// TwinCAT 3 PLC project PLC1
// ProgramVersion: 3.1.4023.0
// libraries:
//   CmpBitmapPool, * (System)
//   Tc2_MC2, * (Beckhoff Automation GmbH)
//   Tc2_Standard, * (Beckhoff Automation GmbH)
//   Tc2_System, * (Beckhoff Automation GmbH)
//   Tc2_Utilities, * (Beckhoff Automation GmbH)
//   Tc3_Module, * (Beckhoff Automation GmbH)
//   VisuDialogs, * (System)
//   VisuSymbols,3.5.10.0,System
// project tree:
//   DUTs/GVLs/ GVL.TcGVL, IOs.TcGVL
//   DUTs/ ST_CSV_Record.TcDUT
//   / GlobalTextList.TcGTLO, PlcTask.TcTTO, VISU_TASK.TcTTO
//   POUs/ Alarmes.TcPOU, InterfaceIOs.TcPOU, MAIN.TcPOU, CondicoesIniciais.TcPOU, IHM.TcPOU, Sinalizadores.TcPOU
//   POUs/Perifericos/ ReguaPotenciometrica.TcPOU, Robo.TcPOU, Inversores.TcPOU, Camera.TcPOU, MaquinaSolda.TcPOU, SafetyPLC.TcPOU, Servos.TcPOU, Valvulas.TcPOU
//   POUs/Receita/ Main_Receita.TcPOU, P_Read_Tabela.TcPOU, P_Write_Tabela.TcPOU
//   VISUs/ ImagePool.TcIPO (not stored), Lista_PontosSolda.TcVIS, Lista_PontosRoboCamera.TcVIS, Tela_Alarmes_2.TcVIS, Tela_Manual_2.TcVIS, Tela_Manual_3.TcVIS, Tela_Alarmes_1.TcVIS, Tela_Producao.TcVIS, Tela_Manual_1.TcVIS, Tela_Receita.TcVIS, Tela_Manutencao.TcVIS, VisualizationManager.TcVMO (not stored)

CONFIGURATION PLC1
    RESOURCE PLC ON TwinCAT3
        TASK PlcTask(INTERVAL := T#10ms, PRIORITY := 10);
        TASK VISU_TASK(INTERVAL := T#200000us, PRIORITY := 30);
        PROGRAM MAIN WITH PlcTask : MAIN;
        PROGRAM VisuElems_Visu_Prg WITH VISU_TASK : VisuElems.Visu_Prg;
    END_RESOURCE
END_CONFIGURATION

// ---- DUTs/ST_CSV_Record.TcDUT
TYPE ST_CSV_Record :
STRUCT
	sName 	: T_MaxString 	:= '';
	nNumber	: UDINT 		:= 0;
	fPos		: LREAL 		:= 0.0;
	bOP		: BOOL 		:= FALSE;
	sDesc		: STRING(40)	:= '';
	data		: ARRAY[0..7] OF BYTE;
END_STRUCT
END_TYPE

// ---- DUTs/GVLs/GVL.TcGVL
VAR_GLOBAL
(*========================================================================*)	

	FB_HoraAtual	: NT_GetTime;
	TempoAtual		: DT;
	Tempo_Atual_UTC	: DT;
	tempo			: TIMESTRUCT;
	
	MaquinaAlarme			: BOOL;
	MaquinaLigada			: BOOL;
	MaquinaModoManual		: BOOL;
	MaquinaModoAuto			: BOOL;
	Flag_CondicoesIniciais	: BOOL;
	Reset					: BOOL;

(*========================================================================*)

(*===================		ENTRADAS DIGITAIS		======================*)
	
	InMaquinaSolda_FK		: BOOL;
	InPinoCalha				: BOOL;
	InReset					: BOOL;
	InVermelho				: BOOL;
	InAmarelo				: BOOL;
	InVerde					: BOOL;
	InPecaOK				: BOOL;
	InSolda					: BOOL;
	
	//Sensores Fins de Curso
	InFimCurso1				: BOOL;
	InFimCurso2				: BOOL;
	InFimCurso3				: BOOL;
	InFimCurso4				: BOOL;

	//Sensores Painel Pneumático
	InPressostatoGeral		: BOOL;
	InSensorSegValvY7 		: BOOL;
	InSensorSegValvY8		: BOOL;
	
	//Sensores Indutivos
	InSensorIndutivo01		: BOOL;
	InSensorIndutivo02		: BOOL;
	InSensorIndutivo03		: BOOL;
	InSensorIndutivo04		: BOOL;
	InSensorIndutivo05		: BOOL;
	InSensorIndutivo06		: BOOL;
	InSensorIndutivo07		: BOOL;
	InSensorIndutivo08		: BOOL;
	InSensorIndutivo09		: BOOL;
	InSensorIndutivo10		: BOOL;
	InSensorIndutivo11		: BOOL;
	InSensorIndutivo12		: BOOL;
	
	//Comandos
	InComandoX				: BOOL;
	InComandoY				: BOOL;
	InComandoZ				: BOOL;
	InComando4				: BOOL;
	InComando5				: BOOL;
	InComando6				: BOOL;
	InComandoX1				: BOOL;
	InComandoX10			: BOOL;
	InComandoX100			: BOOL;
	InComandoStopC			: BOOL;
	InComandoStopCN			: BOOL;
	
	InSinalFaltaFase		: BOOL;
	InComandoPedal			: BOOL;
	InSolicitaEntrada		: BOOL;
	InSolicitaReset			: BOOL;
	
(*========================================================================*)

(*=====================		SAÍDAS DIGITAIS		==========================*)

	//Inversor 1 - Mesa Index
	OutLigarMesaIndex 			: BOOL;
	OutSentidoGiroMesaIndex 	: BOOL;
	
	//Inversor 2 - Esteira de Saída
	OutLigarEsteiraSaida		: BOOL;
	OutSentidoGiroEsteiraSaida	: BOOL;
	
	//Máquina de Solda
	OutMaquinaSolda_BtReset		: BOOL;
	OutMaquinaSolda_BtStart		: BOOL;
	
	OutMaquinaSolda_Receita_Bit1 : BOOL;
	OutMaquinaSolda_Receita_Bit2 : BOOL;
	OutMaquinaSolda_Receita_Bit3 : BOOL;
	OutMaquinaSolda_Receita_Bit4 : BOOL;
	OutMaquinaSolda_Receita_Bit5 : BOOL;
	
	//Válvulas
	OutValvulaY1A				: BOOL;
	OutValvulaY1R				: BOOL;
	OutValvulaY2A				: BOOL;
	OutValvulaY2R				: BOOL;
	OutValvulaY3A				: BOOL;
	OutValvulaY3R				: BOOL;
	OutValvulaY4A				: BOOL;
	OutValvulaY4R				: BOOL;
	OutValvulaY5A				: BOOL;
	OutValvulaY5R				: BOOL;
	OutValvulaY6				: BOOL;
	OutValvulaY7				: BOOL;
	OutValvulaY8				: BOOL;
	OutValvulaY9				: BOOL;
	
	//Sinalizadores Luminosos
	OutSinalizadorComandoLigado	: BOOL;
	OutSinalizadorBotoeiraHS1	: BOOL;
	OutSinalizadorBotoeiraHS2	: BOOL;
	
	//Sinalizador Luminoso - Manivela Eletrônica
	OutSinalizadorManivelaEletronica :BOOL;
	
(*========================================================================*)

(*=========================		SAFETY PLC		==========================*)	

	InSafety_CortinaLuz					: BOOL;
	InSafety_BtEmergenciaMaquinaSolda	: BOOL;
	InSafety_BtEmergenciaChiller		: BOOL;
	InSafety_BtEmergenciaRobo			: BOOL;
	InSafety_BtEmergenciaFrontal		: BOOL;
	InSafety_ChPortaMaquinaSolda		: BOOL;
	InSafety_ChPortaPainelPrincipal		: BOOL;
	InSafety_ChPortaEsteira				: BOOL;
	InSafety_ChPortaCamera				: BOOL;
	InSafety_ChPortaFrontalInferior		: BOOL;
	InSafety_ChPortaLateralEsquerdaFD	: BOOL;
	InSafety_ChPortaLateralEsquerdaFE	: BOOL;
	
	OutSafety_LiberacaoSDV1				: BOOL;
	OutSafety_ComandoSDV1				: BOOL;
	OutSafety_LiberacaoSDV2				: BOOL;
	OutSafety_ComandoSDV2				: BOOL;
	OutSafety_ComandoINVMesaIndex		: BOOL;
	OutSafety_ComandoINVEsteiraSaida	: BOOL;
	OutSafety_Comando1Robo				: BOOL;
	OutSafety_Comando2Robo				: BOOL;
	OutSafety_ParadaMaquinaSolda		: BOOL;
	OutSafety_SinalizacaoEmergencia		: BOOL;
	OutSafety_Reserva1					: BOOL;
	OutSafety_Reserva2					: BOOL;
	
	OutSafety_BtReset					: BOOL;
	
(*========================================================================*)

(*==========================		FLAG's		==========================*)	

	Flag_Maquina_MesaIndex			: BOOL;
	Flag_MesaIndex_Maquina			: BOOL;
	
	Flag_Maquina_EsteiraSaida		: BOOL;
	Flag_EsteiraSaida_Maquina		: BOOL;
	
	//Flag_Maquina_MaquinaSolda		: BOOL;
	//Flag_MaquinaSolda_Maquina		: BOOL;
	Flag_ServosXY_MaquinaSolda		: BOOL;
	Flag_MaquinaSolda_ServosXY		: BOOL;
	
	Flag_Maquina_Robo				: BOOL;
	Flag_Robo_Maquina				: BOOL;
	
	Flag_Robo_Camera				: BOOL;
	Flag_Camera_Robo				: BOOL;
	
	Flag_Maquina_ServosXY			: BOOL;
	Flag_ServosXY_Maquina			: BOOL;

(*========================================================================*)

(*=====================		MÁQUINA DE SOLDA		======================*)	

	LigarMaquinaSoldaManual			: BOOL;
	LigarMaquinaSoldaAuto			: BOOL;

(*========================================================================*)

(*=========================		CÂMERA SICK		==========================*)	

 Camera_Trigger					: BOOL;
 Camera_ChangeJob				: BOOL;
 Camera_SetJob					: BYTE;
 
 Camera_JobResult				: BOOL;
 Camera_JobCompleted			: BOOL;
 Camera_JobID					: BYTE;
 
 PecaAprovada					: BOOL;
 
 Camera_TargetJob				: ARRAY[0..5] OF INT;
 Camera_indexJob				: INT;
 
(*========================================================================*)

(*=========================		ROBÔ YASKAWA	==========================*)	

	Robot_CallMasterJob			: BOOL;
	Robot_ServoOn				: BOOL;
	Robot_ServoOff				: BOOL;
	Robot_ExtStart				: BOOL;
	Robot_ResetAlarm			: BOOL;
	
	Robot_HomePosition			: BOOL;
	Robot_TopMasterJob			: BOOL;
	Robot_AlarmStatus			: BOOL;
	
	
	Robot_IniciarCiclo			: BOOL;
	Robot_JobCompleted			: BOOL;
	Robot_JobCamera				: BOOL;
	
	Robot_NotSafetyPosition		: BOOL;
	
	Robot_Peca					: BOOL;
	Robot_Foto1					: BOOL;
	Robot_Foto2					: BOOL;

(*========================================================================*)

(*======================		SERVO MOTORES		======================*)	

	EixoX 							: AXIS_REF;
	EixoX_Energizado				: BOOL;
	
	EixoY 							: AXIS_REF;
	EixoY_Energizado				: BOOL;

(*========================================================================*)

(*=========================		INVERSORES		==========================*)	

	LigarMesaIndexAutomatico	: BOOL;
	LigarMesaIndexCiclo			: BOOL;
	LigarMesaIndexFwd			: BOOL;
	LigarMesaIndexBwd	 		: BOOL;
	LigarEsteiraSaidaFwd		: BOOL;
	LigarEsteiraSaidaBwd		: BOOL;
	
	FrequenciaMesaIndex			: REAL;
	FrequenciaEsteiraSaida		: REAL;
	
(*========================================================================*)
	
(*=========================		VÁLVULAS		==========================*)	

	AvancarValvulaY1			: BOOL;
	AvancarValvulaY2			: BOOL;
	AvancarValvulaY3			: BOOL;
	AvancarValvulaY4			: BOOL;
	AvancarValvulaY5			: BOOL;
	
	LigarValvulaY6				: BOOL;
	LigarValvulaY7				: BOOL;
	LigarValvulaY8				: BOOL;
	LigarValvulaY9				: BOOL;
	
	ValvulaProporcional			: REAL;
	
(*========================================================================*)

(*======================		ENTRADAS IHM		======================*)

	database_read					: ARRAY[0..MAX_CSV_ROWS, 0..MAX_CSV_COLUMNS ] OF STRING(MAX_CSV_FIELD_LENGTH);(* Target PLC database *)
	Simbolo_Atualizacao				: BOOL;

	b_selecionar_receita			: BOOL;
	b_deletar_receita				: BOOL;
	b_editar_receita				: BOOL;
	b_executar_receita				: BOOL;
	b_salvar_receita				: BOOL;
	b_cancelar_receita				: BOOL;
	b_criar_receita					: BOOL;
	bRead							: BOOL;
	bWrite							: BOOL;
	
(*======================		TELA RECEITA		======================*)

	//IhmEscr_Receita_MaquinaSolda		: INT;

(*======================		TELA MANUAL 1		======================*)
	//Controle da Máquina
	IhmBt_ManualAuto					: BOOL;
	IhmBt_ManualAuto_Text				: STRING;
	IhmBt_ManualAuto_Color				: BOOL;
		
	//ELEMENTOS PNEUMÁTICOS
	IhmBt_Y1_Ligar						: BOOL;
	IhmBt_Y2_Ligar						: BOOL;
	IhmBt_Y3_Ligar						: BOOL;
	IhmBt_Y4_Ligar						: BOOL;
	IhmBt_Y5_Ligar						: BOOL;
	
	IhmBt_Y6_Ligar						: BOOL;
	IhmBt_Y7_Ligar						: BOOL;
	IhmBt_Y8_Ligar						: BOOL;
	IhmBt_Y9_Ligar						: BOOL;	
	
	IhmBt_VP_Teste						: BOOL;
	
	//MOTORES
	//SERVO EIXO X E Y
	IhmBt_ServoXY_X1					: BOOL;
	IhmBt_ServoXY_X10					: BOOL;
	IhmBt_ServoXY_X100					: BOOL;
	
	//SERVO EIXO X
	IhmBt_ServoX_Reset					: BOOL;
	IhmBt_ServoX_Home					: BOOL;
	IhmBt_ServoX_JogBwd					: BOOL;
	IhmBt_ServoX_JogFwd					: BOOL;
	IhmBt_ServoX_PowerOn				: BOOL;
	IhmBt_ServoX_Referenciar			: BOOL;
	
	IhmLeit_ServoX_Posicao				: LREAL;
	IhmLeit_ServoX_Velocidade			: LREAL;
	IhmLeit_ServoX_Torque				: LREAL;
	
	//SERVO EIXO Y
	IhmBt_ServoY_Reset					: BOOL;
	IhmBt_ServoY_Home					: BOOL;
	IhmBt_ServoY_JogBwd					: BOOL;
	IhmBt_ServoY_JogFwd					: BOOL;
	IhmBt_ServoY_PowerOn				: BOOL;
	IhmBt_ServoY_Referenciar			: BOOL;
		
	IhmLeit_ServoY_Posicao				: LREAL;
	IhmLeit_ServoY_Velocidade			: LREAL;
	IhmLeit_ServoY_Torque				: LREAL;
	
	//INV. MESA INDEX
	IhmBt_MesaIndex_Sentido				: BOOL;
	IhmBt_MesaIndex_LigarDesligar		: BOOL;
	IhmBt_MesaIndex_Ciclo				: BOOL;
	
	//INV. ESTEIRA DE SAÍDA
	IhmBt_EsteiraSaida_Sentido			: BOOL;
	IhmBt_EsteiraSaida_LigarDesligar	: BOOL;
	
	IhmBt_MaquinaSolda_Reset			: BOOL;
	IhmBt_MaquinaSolda_Start			: BOOL;

(*======================		TELA MANUAL 2		======================*)
	
	IhmBt_ServoX_ReferenciarAutoINICIO				: BOOL;
	IhmBt_ServoX_ReferenciarAutoFIM					: BOOL;
	IhmBt_ServoY_ReferenciarAutoINICIO				: BOOL;
	IhmBt_ServoY_ReferenciarAutoFIM					: BOOL;
	
	IhmVs_PressaoPainelPneumatico_Text				: WSTRING;
	
	IhmBt_ReguaPotenciometrica_CalibrarRecuo		: BOOL;
	IhmBt_ReguaPotenciometrica_CalibrarPorca		: BOOL;
	IhmBt_ReguaPotenciometrica_CalibrarAvanco		: BOOL;
		
(*======================		TELA MANUAL 3		======================*)
	
	IhmBt_Camera_ChangeJob					: BOOL;
	IhmBt_Camera_Trigger					: BOOL;
	IhmLed_Camera_JobCompleted				: BOOL;
	IhmLed_Camera_JobResult					: BOOL;
	
	IhmLeit_Camera_JobID					: INT;
	
	IhmVs_Camera_JobResult_Text				: STRING;
		
(*========================================================================*)
	
	UserName		: STRING;
	UserGroupName	: STRING;
	UserGroupId		: DWORD;
	
	Blink_1hz		: BOOL;
	Blick_05hz		: BOOL;
	
	IhmBt_Ligar			: BOOL;
	IhmBt_Desligar		: BOOL;
	IhmBt_Reset			: BOOL;
	IhmBt_Pausar		: BOOL;
	IhmBt_CondIniciais	: BOOL;
	
	BT_ihm_zerar_contador	: BOOL;
	Contador_Total			: UDINT;
	Contador_PecasAprovadas	: UDINT;
	Contador_PecasReprovadas: UDINT;
	
	I1		: BOOL;
	I2		: BOOL;
	
	Recipe_Select_Int				: UDINT;
	Recipe_Names_Saved				: ARRAY [0..301] OF STRING;
	
	Recipe_Name_Select				: STRING;
	
	Recipe_No_Select				: INT;
	Recipe_ID_Select				: INT;
	
//	Recipe_Pos_HomeX_Select			: LREAL;
//	Recipe_Pos_HomeY_Select			: LREAL;
	
	Recipe_Pontos_Solda_Select		: INT;
	
	Recipe_P_X01_Solda_Select		: LREAL;
	Recipe_P_Y01_Solda_Select		: LREAL;
	Recipe_P01_Solda_Select			: BOOL;
	
	Recipe_P_X02_Solda_Select		: LREAL;
	Recipe_P_Y02_Solda_Select		: LREAL;
	Recipe_P02_Solda_Select			: BOOL;
	
	Recipe_P_X03_Solda_Select		: LREAL;
	Recipe_P_Y03_Solda_Select		: LREAL;
	Recipe_P03_Solda_Select			: BOOL;
	
	Recipe_P_X04_Solda_Select		: LREAL;
	Recipe_P_Y04_Solda_Select		: LREAL;
	Recipe_P04_Solda_Select			: BOOL;
	
	Recipe_P_X05_Solda_Select		: LREAL;
	Recipe_P_Y05_Solda_Select		: LREAL;
	Recipe_P05_Solda_Select			: BOOL;
	
	Recipe_P_X06_Solda_Select		: LREAL;
	Recipe_P_Y06_Solda_Select		: LREAL;
	Recipe_P06_Solda_Select			: BOOL;
	
	Recipe_P_X07_Solda_Select		: LREAL;
	Recipe_P_Y07_Solda_Select		: LREAL;
	Recipe_P07_Solda_Select			: BOOL;
	
	Recipe_P_X08_Solda_Select		: LREAL;
	Recipe_P_Y08_Solda_Select		: LREAL;
	Recipe_P08_Solda_Select			: BOOL;
	
	Recipe_P_X09_Solda_Select		: LREAL;
	Recipe_P_Y09_Solda_Select		: LREAL;
	Recipe_P09_Solda_Select			: BOOL;
	
	Recipe_P_X10_Solda_Select		: LREAL;
	Recipe_P_Y10_Solda_Select		: LREAL;
	Recipe_P10_Solda_Select			: BOOL;
	
	Recipe_P_X11_Solda_Select		: LREAL;
	Recipe_P_Y11_Solda_Select		: LREAL;
	Recipe_P11_Solda_Select			: BOOL;
	
	Recipe_P_X12_Solda_Select		: LREAL;
	Recipe_P_Y12_Solda_Select		: LREAL;
	Recipe_P12_Solda_Select			: BOOL;
	
	Recipe_P_X13_Solda_Select		: LREAL;
	Recipe_P_Y13_Solda_Select		: LREAL;
	Recipe_P13_Solda_Select			: BOOL;
	
	Recipe_P_X14_Solda_Select		: LREAL;
	Recipe_P_Y14_Solda_Select		: LREAL;
	Recipe_P14_Solda_Select			: BOOL;
	
	Recipe_P_X15_Solda_Select		: LREAL;
	Recipe_P_Y15_Solda_Select		: LREAL;
	Recipe_P15_Solda_Select			: BOOL;

	Recipe_Pontos_Camera_Select		: INT;
	Recipe_JobID_F01_Camera_Select	: INT;
	Recipe_JobID_F02_Camera_Select	: INT;
	Recipe_JobID_F03_Camera_Select	: INT;
	Recipe_JobID_F04_Camera_Select	: INT;
	Recipe_JobID_F05_Camera_Select	: INT;
	
//	Recipe_F01_Camera_Select		: BOOL;
//	Recipe_F02_Camera_Select		: BOOL;
//	Recipe_F03_Camera_Select		: BOOL;
//	Recipe_F04_Camera_Select		: BOOL;
//	Recipe_F05_Camera_Select		: BOOL;


	Recipe_Valvula_Proporcional_Select	: LREAL;
	
	Recipe_Pecas_Caixa_Select		: INT;
		
	NumPontosSolda					: INT;
	NumPontosCamera					: INT;
	
	TargetX							: ARRAY[0..14] OF LREAL;
	TargetY							: ARRAY[0..14] OF LREAL;
	SoldaXY							: ARRAY[0..14] OF BOOL;
	
	CameraJobID						: ARRAY[0..4] OF INT;
	
	PosicaoOrigemX					: LREAL;
	PosicaoOrigemY					: LREAL;
	
(*========================================================================*)
	
END_VAR

VAR_GLOBAL RETAIN

(*======================		TELA RECEITA		======================*)

	IhmEscr_Receita_MaquinaSolda		: INT;

(*======================		TELA MANUAL 1		======================*)

	//ELEMENTOS PNEUMÁTICOS
	IhmEscr_ValvulaProporcional			: INT;

	//SERVO EIXO X E Y
	IhmEscr_ServoXY_TorqueMax			: INT;
	IhmEscr_ServoXY_TempoTorqueMax		: INT;
	IhmEscr_ServoXY_VelocidadeAuto		: INT;
	IhmEscr_ServoXY_VelocidadeManual	: INT;
	
	//INV. MESA INDEX
	IhmEscr_MesaIndex_Frequencia		: INT;
	IhmEscr_MesaIndex_DelayParada		: REAL;
	
	//INV. ESTEIRA DE SAÍDA
	IhmEscr_EsteiraSaida_Frequencia		: INT;

(*======================		TELA MANUAL 2		======================*)
	
	IhmEscr_ReguaPotenciometrica_ToleranciaRecuo	: REAL;
	IhmEscr_ReguaPotenciometrica_ToleranciaPorca	: REAL;
	IhmEscr_ReguaPotenciometrica_ToleranciaAvanco	: REAL;	
		
(*======================		TELA MANUAL 3		======================*)
	
	IhmEscr_Camera_SetJob					: INT;
	
	IhmEscr_Camera_DelayError				: TIME;
	
(*==================		RÉGUA POTENCIOMÉTRICA		==================*)	

	ReguaPotenciometricaPosicao			: REAL;
	ReguaPotenciometricaSinal			: INT;
	
	ReguaPotenciometrica_Recuada		: REAL;
	ReguaPotenciometrica_Recuada_LI		: REAL;
	ReguaPotenciometrica_Recuada_LS		: REAL;

	ReguaPotenciometrica_Porca			: REAL;
	ReguaPotenciometrica_Porca_LI		: REAL;
	ReguaPotenciometrica_Porca_LS		: REAL;

	ReguaPotenciometrica_Avancada		: REAL;
	ReguaPotenciometrica_Avancada_LI	: REAL;
	ReguaPotenciometrica_Avancada_LS	: REAL;
	
(*========================================================================*)

END_VAR

VAR_GLOBAL CONSTANT

	MAX_CSV_ROWS 			: UDINT := 30;
	MAX_CSV_COLUMNS 		: UDINT := 60;
	MAX_CSV_FIELD_LENGTH	: UDINT := 100;

END_VAR

// ---- DUTs/GVLs/IOs.TcGVL
VAR_GLOBAL

(*======================		ENTRADAS DIGITAIS		======================*)

	//Cartão de Entradas 0:= EntradaI0_0
	EntradaI0_0		AT %I*	: BOOL;
	EntradaI0_1		AT %I*	: BOOL;
	EntradaI0_2		AT %I*	: BOOL;
	EntradaI0_3		AT %I*	: BOOL;
	EntradaI0_4		AT %I*	: BOOL;
	EntradaI0_5		AT %I*	: BOOL;
	EntradaI0_6		AT %I*	: BOOL;
	EntradaI0_7		AT %I*	: BOOL;
	EntradaI1_0		AT %I*	: BOOL;
	EntradaI1_1		AT %I*	: BOOL;
	EntradaI1_2		AT %I*	: BOOL;
	EntradaI1_3		AT %I*	: BOOL;
	EntradaI1_4		AT %I*	: BOOL;
	EntradaI1_5		AT %I*	: BOOL;
	EntradaI1_6		AT %I*	: BOOL;
	EntradaI1_7		AT %I*	: BOOL;
	
	//Cartão de Entradas 1
	EntradaI2_0		AT %I*	: BOOL;
	EntradaI2_1		AT %I*	: BOOL;
	EntradaI2_2		AT %I*	: BOOL;
	EntradaI2_3		AT %I*	: BOOL;
	EntradaI2_4		AT %I*	: BOOL;
	EntradaI2_5		AT %I*	: BOOL;
	EntradaI2_6		AT %I*	: BOOL;
	EntradaI2_7		AT %I*	: BOOL;
	EntradaI3_0		AT %I*	: BOOL;
	EntradaI3_1		AT %I*	: BOOL;
	EntradaI3_2		AT %I*	: BOOL;
	EntradaI3_3		AT %I*	: BOOL;
	EntradaI3_4		AT %I*	: BOOL;
	EntradaI3_5		AT %I*	: BOOL;
	EntradaI3_6		AT %I*	: BOOL;
	EntradaI3_7		AT %I*	: BOOL;
	
	//Cartão de Entradas 2
	EntradaI4_0		AT %I*	: BOOL;
	EntradaI4_1		AT %I*	: BOOL;
	EntradaI4_2		AT %I*	: BOOL;
	EntradaI4_3		AT %I*	: BOOL;
	EntradaI4_4		AT %I*	: BOOL;
	EntradaI4_5		AT %I*	: BOOL;
	EntradaI4_6		AT %I*	: BOOL;
	EntradaI4_7		AT %I*	: BOOL;
	EntradaI5_0		AT %I*	: BOOL;
	EntradaI5_1		AT %I*	: BOOL;
	EntradaI5_2		AT %I*	: BOOL;
	EntradaI5_3		AT %I*	: BOOL;
	EntradaI5_4		AT %I*	: BOOL;
	EntradaI5_5		AT %I*	: BOOL;
	EntradaI5_6		AT %I*	: BOOL;
	EntradaI5_7		AT %I*	: BOOL;
	
	//Cartão de Entradas 3
	EntradaI6_0		AT %I*	: BOOL;
	EntradaI6_1		AT %I*	: BOOL;
	EntradaI6_2		AT %I*	: BOOL;
	EntradaI6_3		AT %I*	: BOOL;
	EntradaI6_4		AT %I*	: BOOL;
	EntradaI6_5		AT %I*	: BOOL;
	EntradaI6_6		AT %I*	: BOOL;
	EntradaI6_7		AT %I*	: BOOL;
	EntradaI7_0		AT %I*	: BOOL;
	EntradaI7_1		AT %I*	: BOOL;
	EntradaI7_2		AT %I*	: BOOL;
	EntradaI7_3		AT %I*	: BOOL;
	EntradaI7_4		AT %I*	: BOOL;
	EntradaI7_5		AT %I*	: BOOL;
	EntradaI7_6		AT %I*	: BOOL;
	EntradaI7_7		AT %I*	: BOOL;
	
(*============================================================================*)
(*=========================		SAÍDAS DIGITAIS		==========================*)
	//Outputs
	
	//Cartão de Saídas 0
	SaidaQ0_0		AT %Q*	: BOOL;
	SaidaQ0_1		AT %Q*	: BOOL;
	SaidaQ0_2		AT %Q*	: BOOL;
	SaidaQ0_3		AT %Q*	: BOOL;
	SaidaQ0_4		AT %Q*	: BOOL;
	SaidaQ0_5		AT %Q*	: BOOL;
	SaidaQ0_6		AT %Q*	: BOOL;
	SaidaQ0_7		AT %Q*	: BOOL;
	SaidaQ1_0		AT %Q*	: BOOL;
	SaidaQ1_1		AT %Q*	: BOOL;
	SaidaQ1_2		AT %Q*	: BOOL;
	SaidaQ1_3		AT %Q*	: BOOL;
	SaidaQ1_4		AT %Q*	: BOOL;
	SaidaQ1_5		AT %Q*	: BOOL;
	SaidaQ1_6		AT %Q*	: BOOL;
	SaidaQ1_7		AT %Q*	: BOOL;
	
	//Cartão de Saídas 1
	SaidaQ2_0		AT %Q*	: BOOL;
	SaidaQ2_1		AT %Q*	: BOOL;
	SaidaQ2_2		AT %Q*	: BOOL;
	SaidaQ2_3		AT %Q*	: BOOL;
	SaidaQ2_4		AT %Q*	: BOOL;
	SaidaQ2_5		AT %Q*	: BOOL;
	SaidaQ2_6		AT %Q*	: BOOL;
	SaidaQ2_7		AT %Q*	: BOOL;
	SaidaQ3_0		AT %Q*	: BOOL;
	SaidaQ3_1		AT %Q*	: BOOL;
	SaidaQ3_2		AT %Q*	: BOOL;
	SaidaQ3_3		AT %Q*	: BOOL;
	SaidaQ3_4		AT %Q*	: BOOL;
	SaidaQ3_5		AT %Q*	: BOOL;
	SaidaQ3_6		AT %Q*	: BOOL;
	SaidaQ3_7		AT %Q*	: BOOL;
	
	//Cartão de Saídas 2
	SaidaQ4_0		AT %Q*	: BOOL;
	SaidaQ4_1		AT %Q*	: BOOL;
	SaidaQ4_2		AT %Q*	: BOOL;
	SaidaQ4_3		AT %Q*	: BOOL;
	SaidaQ4_4		AT %Q*	: BOOL;
	SaidaQ4_5		AT %Q*	: BOOL;
	SaidaQ4_6		AT %Q*	: BOOL;
	SaidaQ4_7		AT %Q*	: BOOL;
	SaidaQ5_0		AT %Q*	: BOOL;
	SaidaQ5_1		AT %Q*	: BOOL;
	SaidaQ5_2		AT %Q*	: BOOL;
	SaidaQ5_3		AT %Q*	: BOOL;
	SaidaQ5_4		AT %Q*	: BOOL;
	SaidaQ5_5		AT %Q*	: BOOL;
	SaidaQ5_6		AT %Q*	: BOOL;
	SaidaQ5_7		AT %Q*	: BOOL;
	
	//Cartão de Saídas 3
	SaidaQ6_0		AT %Q*	: BOOL;
	SaidaQ6_1		AT %Q*	: BOOL;
	SaidaQ6_2		AT %Q*	: BOOL;
	SaidaQ6_3		AT %Q*	: BOOL;
	SaidaQ6_4		AT %Q*	: BOOL;
	SaidaQ6_5		AT %Q*	: BOOL;
	SaidaQ6_6		AT %Q*	: BOOL;
	SaidaQ6_7		AT %Q*	: BOOL;
	SaidaQ7_0		AT %Q*	: BOOL;
	SaidaQ7_1		AT %Q*	: BOOL;
	SaidaQ7_2		AT %Q*	: BOOL;
	SaidaQ7_3		AT %Q*	: BOOL;
	SaidaQ7_4		AT %Q*	: BOOL;
	SaidaQ7_5		AT %Q*	: BOOL;
	SaidaQ7_6		AT %Q*	: BOOL;
	SaidaQ7_7		AT %Q*	: BOOL;	

(*============================================================================*)
(*======================		ENTRADAS ANALÓGICAS		======================*)

	//Cartão de Entradas
	EntradaA0_0		AT %I*	: INT;
	EntradaA0_1		AT %I*	: INT;
	EntradaA0_2		AT %I*	: INT;
	EntradaA0_3		AT %I*	: INT;

(*============================================================================*)	
	
(*============================================================================*)
(*======================		SAÍDAS ANALÓGICAS		======================*)

	//Cartão de Saídas 0
	SaidaA0_0		AT %Q*	: INT;
	SaidaA0_1		AT %Q*	: INT;
	SaidaA0_2		AT %Q*	: INT;
	SaidaA0_3		AT %Q*	: INT;
		
(*============================================================================*)

(*======================		REDE ETHERNET/IP		======================*)

(*==========================		SAFETY PLC		==========================*)

	SafetyPLC_In_Byte0 		AT %I*:BYTE;
	SafetyPLC_In_Byte1 		AT %I*:BYTE;
	SafetyPLC_In_Byte2 		AT %I*:BYTE;
	SafetyPLC_In_Byte3 		AT %I*:BYTE;
	SafetyPLC_In_Byte4 		AT %I*:BYTE;
	SafetyPLC_In_Byte5 		AT %I*:BYTE;
	
	SafetyPLC_Out_Byte0 	AT %Q*:BYTE;

(*============================================================================*)

(*===================		CÂMERA SICK - INSPECTOR 63		==================*)

	CameraSickIn_0		AT %I*:BYTE;
	CameraSickIn_1		AT %I*:BYTE;
	CameraSickIn_2		AT %I*:BYTE;
	CameraSickIn_3		AT %I*:BYTE;
	CameraSickIn_4		AT %I*:BYTE;
	CameraSickIn_5		AT %I*:BYTE;
	CameraSickIn_6		AT %I*:BYTE;
	CameraSickIn_7		AT %I*:BYTE;
	CameraSickIn_8		AT %I*:BYTE;
	CameraSickIn_9		AT %I*:BYTE;

	CameraSickOut_0		AT %Q*:BYTE;
	CameraSickOut_1		AT %Q*:BYTE;
	CameraSickOut_2		AT %Q*:BYTE;
	CameraSickOut_3		AT %Q*:BYTE;
	CameraSickOut_4		AT %Q*:BYTE;
	CameraSickOut_5		AT %Q*:BYTE;
	CameraSickOut_6		AT %Q*:BYTE;
	CameraSickOut_7		AT %Q*:BYTE;
	CameraSickOut_8		AT %Q*:BYTE;
	CameraSickOut_9		AT %Q*:BYTE;

(*============================================================================*)

(*=====================		ROBÔ YASKAWA/MOTOMAN		======================*)
	
	Robot_PLC_0 		AT %I*:BYTE;
	Robot_PLC_1 		AT %I*:BYTE;
	Robot_PLC_2 		AT %I*:BYTE;
	Robot_PLC_3 		AT %I*:BYTE;
	Robot_PLC_4 		AT %I*:BYTE;
	Robot_PLC_5 		AT %I*:BYTE;
	Robot_PLC_6 		AT %I*:BYTE;
	Robot_PLC_7 		AT %I*:BYTE;
	Robot_PLC_8 		AT %I*:BYTE;
	Robot_PLC_9 		AT %I*:BYTE;
	Robot_PLC_10 		AT %I*:BYTE;
	Robot_PLC_11 		AT %I*:BYTE;
	Robot_PLC_12 		AT %I*:BYTE;
	Robot_PLC_13 		AT %I*:BYTE;
	Robot_PLC_14 		AT %I*:BYTE;
	Robot_PLC_15 		AT %I*:BYTE;
	Robot_PLC_16 		AT %I*:BYTE;
	Robot_PLC_17 		AT %I*:BYTE;
	Robot_PLC_18 		AT %I*:BYTE;
	Robot_PLC_19 		AT %I*:BYTE;
	
	PLC_Robot_0			AT %Q*:BYTE;
	PLC_Robot_1			AT %Q*:BYTE;
	PLC_Robot_2			AT %Q*:BYTE;
	PLC_Robot_3			AT %Q*:BYTE;
	PLC_Robot_4			AT %Q*:BYTE;
	PLC_Robot_5			AT %Q*:BYTE;
	PLC_Robot_6			AT %Q*:BYTE;
	PLC_Robot_7			AT %Q*:BYTE;
	PLC_Robot_8			AT %Q*:BYTE;
	PLC_Robot_9			AT %Q*:BYTE;
	PLC_Robot_10		AT %Q*:BYTE;
	PLC_Robot_11		AT %Q*:BYTE;
	PLC_Robot_12		AT %Q*:BYTE;
	PLC_Robot_13		AT %Q*:BYTE;
	PLC_Robot_14		AT %Q*:BYTE;
	PLC_Robot_15		AT %Q*:BYTE;

(*============================================================================*)
	
END_VAR

// ---- POUs/MAIN.TcPOU
PROGRAM MAIN
VAR
		
	SafetyPLCIn 	AT %I*:BYTE;
	SafetyPLCOut 	AT %Q*:BYTE;
	
	sUrlAddressCamera : STRING;

	writeData:FB_WritePersistentData;
	t1:TON;
	bSavePersistent: BOOL;
	
	timer_login	: TON;
	
	Timer_Blink_1hz_1	: TON;
	Timer_Blink_1hz_2	: TON;
	
	b_contador		: BOOL;
	int_contador_10		: INT;
	
	
	PassoBtLigarDesligar	: INT;
	PassoBtReset			: INT;
	PassoMaquina			: INT;
	
END_VAR

(*=====================		ROTINAS EXECUTADAS		======================*)

Main_Receita();
CondicoesIniciais();
Alarmes();
InterfaceIOs();
Inversores();
Valvulas();
ReguaPotenciometrica();
Servos();
Robo();
Camera();
MaquinaSolda();
IHM();
Sinalizadores();

(*=================		INTERFACE CÂMERA SICK		======================*)

sUrlAddressCamera := 'http://192.168.10.20/';

(*=====================		ROTINA PRINCIPAL		======================*)	

//Condição de Bloqueio da Máquina de Estados - Mesa Index FWD
IF (Alarmes.AlarmeGrave
	//OR Alarmes.AlarmeMedio
	//OR Alarmes.AlarmeLeve
	OR NOT MaquinaLigada
	OR NOT MaquinaModoAuto
	) THEN
	PassoMaquina := 1000;
	MaquinaLigada := FALSE;
	Flag_Maquina_MesaIndex := FALSE;
	Flag_Maquina_ServosXY := FALSE;	
	Flag_Maquina_Robo := FALSE;
	Flag_Maquina_EsteiraSaida := FALSE;
END_IF

CASE PassoMaquina OF

	//Passo 0 - Inicialização
	0: PassoMaquina := 10;
	
	//Passo 10 - Verificar condições iniciais
	10: PassoMaquina := 20;
	
	//Passo 20 - Comando para iniciar ciclo 
	20: //IF InComandoPedal THEN
			PassoMaquina := 30;
		//END_IF
	
	//Passo 30 - Dar Passo na Mesa Index
	30: Flag_Maquina_MesaIndex := TRUE;
		PassoMaquina := 40;
		
	//Passo 40 - Verificar Conclusão do Movimento da Mesa Index
	40: IF Flag_MesaIndex_Maquina THEN
			Flag_MesaIndex_Maquina := FALSE;
			PassoMaquina := 50;
		END_IF
		
	//Passo 50 - Liberar Servos XY
	50: Flag_Maquina_ServosXY := TRUE;
		PassoMaquina := 60;
		
	//Passo 60 - Liberar Ação do Robô
	60: Flag_Maquina_Robo := TRUE;
		PassoMaquina := 70;
		
	//Passo 70 - Verificar Conclusão da Rotina dos Servos e da Máquina de Solda
	70: IF Flag_ServosXY_Maquina THEN
			Flag_ServosXY_Maquina := FALSE;
			PassoMaquina := 80;
		END_IF
	
	//Passo 80 - Verificar Conclusão da Rotina Avaliação da Peça (Robô e Câmera)
	80: IF Flag_Robo_Maquina THEN
			Flag_Robo_Maquina := FALSE;
			PassoMaquina := 1000;
		END_IF
	
	//Passo 1000 - Finalização
	1000: PassoMaquina := 0;

END_CASE

(*========================================================================*)

END_PROGRAM

// ---- POUs/Receita/Main_Receita.TcPOU
PROGRAM Main_Receita
VAR
	(*	In USA/UK the CSV field separator is a comma.
	In Germany and some other European countries the CSV field separator is a semicolon. *)
	bChangeSeparatorToComma	: BOOL := FALSE;
	
	i : UDINT;
	
	PassoLimparMemoriasReceita 	: INT;
	
	timer_Leitura_Receitas_Salvas	: TON;
	Endereco_vazio		: INT;
	b_reorganizar		: INT;
	Item_deletado		: UDINT;
	Item_criar			: UDINT;
	Item_livre			: UDINT;
	Item_Atual			: UDINT;
	
	Row_copy			: ARRAY[0..MAX_CSV_COLUMNS] OF STRING(MAX_CSV_FIELD_LENGTH);(* Target PLC database *)
	
	LengthScrollBar_PontosSolda			: INT;
	ScrollBar_PontosSolda				: INT;
	ScrollScreen_PontosSolda			: INT;
	
	LengthScrollBar_PontosCamera		: INT;
	ScrollBar_PontosCamera				: INT;
	ScrollScreen_PontosCamera			: INT;
	
END_VAR

(*========================================================================*)
(*=============		BARRA DE ROLAGEM - TELA RECEITAS		==============*)

//Lista de Pontos de Solda
IF(Recipe_Pontos_Solda_Select <=2) THEN
	ScrollBar_PontosSolda := 0;
	LengthScrollBar_PontosSolda := 0;
ELSE
	LengthScrollBar_PontosSolda := (Recipe_Pontos_Solda_Select-2)*60;
END_IF

ScrollScreen_PontosSolda := (-1)*ScrollBar_PontosSolda;

//Lista de Pontos de Avaliação - Câmera
IF(Recipe_Pontos_Camera_Select <=2) THEN
	ScrollBar_PontosCamera := 0;
	LengthScrollBar_PontosCamera := 0;
ELSE
	LengthScrollBar_PontosCamera := (Recipe_Pontos_Camera_Select-2)*60;
END_IF

ScrollScreen_PontosCamera := (-1)*ScrollBar_PontosCamera;

(*========================================================================*)

IF bChangeSeparatorToComma THEN
	DEFAULT_CSV_FIELD_SEP := 16#2C;(* Comma ASCII code *)
ELSE
	DEFAULT_CSV_FIELD_SEP := 16#3B;(* Semicolon ASCII code *)
END_IF

P_Read_Tabela();
P_Write_Tabela();
//P_ArgToConvExample();(* This sample program shows the usage of the ARG_TO_CSVFIELD and CSVFILED_TO_ARG conversion functions *)
//P_StringToConvExample(); (* This sample program shows the usage of the STRING_TO_CSVFIELD and CSVFIELD_TO_STRING conversion functions *)

(*timer_Leitura_Receitas_Salvas (in := TRUE, pt := T#1M);
IF timer_Leitura_Receitas_Salvas.Q THEN
	timer_Leitura_Receitas_Salvas (in := FALSE);
	bRead := TRUE;
END_IF*)

IF NOT b_deletar_receita AND NOT b_editar_receita AND NOT b_criar_receita THEN
	
	Recipe_Name_Select					:= database_read[Recipe_select_int, 0];
	Recipe_No_Select					:= STRING_TO_INT	(database_read[Recipe_select_int, 1]);
	Recipe_ID_Select					:= STRING_TO_INT	(database_read[Recipe_select_int, 2]);
		
	Recipe_Pontos_Solda_Select			:= STRING_TO_INT	(database_read[Recipe_select_int, 3]);
		
	Recipe_P_X01_Solda_Select			:= STRING_TO_LREAL 	(database_read[Recipe_select_int, 4]);
	Recipe_P_Y01_Solda_Select			:= STRING_TO_LREAL 	(database_read[Recipe_select_int, 5]);
	Recipe_P01_Solda_Select				:= STRING_TO_BOOL	(database_read[Recipe_select_int, 6]);
	Recipe_P_X02_Solda_Select			:= STRING_TO_LREAL 	(database_read[Recipe_select_int, 7]);
	Recipe_P_Y02_Solda_Select			:= STRING_TO_LREAL 	(database_read[Recipe_select_int, 8]);
	Recipe_P02_Solda_Select				:= STRING_TO_BOOL	(database_read[Recipe_select_int, 9]);	
	Recipe_P_X03_Solda_Select			:= STRING_TO_LREAL 	(database_read[Recipe_select_int, 10]);
	Recipe_P_Y03_Solda_Select			:= STRING_TO_LREAL 	(database_read[Recipe_select_int, 11]);
	Recipe_P03_Solda_Select				:= STRING_TO_BOOL	(database_read[Recipe_select_int, 12]);
	Recipe_P_X04_Solda_Select			:= STRING_TO_LREAL 	(database_read[Recipe_select_int, 13]);
	Recipe_P_Y04_Solda_Select			:= STRING_TO_LREAL 	(database_read[Recipe_select_int, 14]);
	Recipe_P04_Solda_Select				:= STRING_TO_BOOL	(database_read[Recipe_select_int, 15]);
	Recipe_P_X05_Solda_Select			:= STRING_TO_LREAL 	(database_read[Recipe_select_int, 16]);
	Recipe_P_Y05_Solda_Select			:= STRING_TO_LREAL 	(database_read[Recipe_select_int, 17]);
	Recipe_P05_Solda_Select				:= STRING_TO_BOOL	(database_read[Recipe_select_int, 18]);
	
	Recipe_P_X06_Solda_Select			:= STRING_TO_LREAL 	(database_read[Recipe_select_int, 19]);
	Recipe_P_Y06_Solda_Select			:= STRING_TO_LREAL 	(database_read[Recipe_select_int, 20]);
	Recipe_P06_Solda_Select				:= STRING_TO_BOOL	(database_read[Recipe_select_int, 21]);
	Recipe_P_X07_Solda_Select			:= STRING_TO_LREAL 	(database_read[Recipe_select_int, 22]);
	Recipe_P_Y07_Solda_Select			:= STRING_TO_LREAL 	(database_read[Recipe_select_int, 23]);
	Recipe_P07_Solda_Select				:= STRING_TO_BOOL	(database_read[Recipe_select_int, 24]);	
	Recipe_P_X08_Solda_Select			:= STRING_TO_LREAL 	(database_read[Recipe_select_int, 25]);
	Recipe_P_Y08_Solda_Select			:= STRING_TO_LREAL 	(database_read[Recipe_select_int, 26]);
	Recipe_P08_Solda_Select				:= STRING_TO_BOOL	(database_read[Recipe_select_int, 27]);
	Recipe_P_X09_Solda_Select			:= STRING_TO_LREAL 	(database_read[Recipe_select_int, 28]);
	Recipe_P_Y09_Solda_Select			:= STRING_TO_LREAL 	(database_read[Recipe_select_int, 29]);
	Recipe_P09_Solda_Select				:= STRING_TO_BOOL	(database_read[Recipe_select_int, 30]);
	Recipe_P_X10_Solda_Select			:= STRING_TO_LREAL 	(database_read[Recipe_select_int, 31]);
	Recipe_P_Y10_Solda_Select			:= STRING_TO_LREAL 	(database_read[Recipe_select_int, 32]);
	Recipe_P10_Solda_Select				:= STRING_TO_BOOL	(database_read[Recipe_select_int, 33]);
		
	Recipe_P_X11_Solda_Select			:= STRING_TO_LREAL 	(database_read[Recipe_select_int, 34]);
	Recipe_P_Y11_Solda_Select			:= STRING_TO_LREAL 	(database_read[Recipe_select_int, 35]);
	Recipe_P11_Solda_Select				:= STRING_TO_BOOL	(database_read[Recipe_select_int, 36]);
	Recipe_P_X12_Solda_Select			:= STRING_TO_LREAL 	(database_read[Recipe_select_int, 37]);
	Recipe_P_Y12_Solda_Select			:= STRING_TO_LREAL 	(database_read[Recipe_select_int, 38]);
	Recipe_P12_Solda_Select				:= STRING_TO_BOOL	(database_read[Recipe_select_int, 39]);	
	Recipe_P_X13_Solda_Select			:= STRING_TO_LREAL 	(database_read[Recipe_select_int, 40]);
	Recipe_P_Y13_Solda_Select			:= STRING_TO_LREAL 	(database_read[Recipe_select_int, 41]);
	Recipe_P13_Solda_Select				:= STRING_TO_BOOL	(database_read[Recipe_select_int, 42]);
	Recipe_P_X14_Solda_Select			:= STRING_TO_LREAL 	(database_read[Recipe_select_int, 43]);
	Recipe_P_Y14_Solda_Select			:= STRING_TO_LREAL 	(database_read[Recipe_select_int, 44]);
	Recipe_P14_Solda_Select				:= STRING_TO_BOOL	(database_read[Recipe_select_int, 45]);
	Recipe_P_X15_Solda_Select			:= STRING_TO_LREAL 	(database_read[Recipe_select_int, 46]);
	Recipe_P_Y15_Solda_Select			:= STRING_TO_LREAL 	(database_read[Recipe_select_int, 47]);
	Recipe_P15_Solda_Select				:= STRING_TO_BOOL	(database_read[Recipe_select_int, 48]);
		
	Recipe_Valvula_Proporcional_Select	:= STRING_TO_LREAL 	(database_read[Recipe_select_int, 49]);
	
	Recipe_Pontos_Camera_Select			:= STRING_TO_INT	(database_read[Recipe_select_int, 50]);
	Recipe_JobID_F01_Camera_Select		:= STRING_TO_INT 	(database_read[Recipe_select_int, 51]);
	Recipe_JobID_F02_Camera_Select		:= STRING_TO_INT 	(database_read[Recipe_select_int, 52]);
	Recipe_JobID_F03_Camera_Select		:= STRING_TO_INT 	(database_read[Recipe_select_int, 53]);
	Recipe_JobID_F04_Camera_Select		:= STRING_TO_INT 	(database_read[Recipe_select_int, 54]);
	Recipe_JobID_F05_Camera_Select		:= STRING_TO_INT 	(database_read[Recipe_select_int, 55]);

	Recipe_Pecas_Caixa_Select			:= STRING_TO_INT 	(database_read[Recipe_select_int, 56]);
	
	Recipe_names_saved [i] := database_read [i,0];

	IF Recipe_names_saved[i] <> '' THEN
		Item_Atual := 1;	
	END_IF
	
	IF Item_Atual = 1 AND Recipe_names_saved[i] = '' THEN
		Item_Atual := 0;
		Item_livre := i;
		i:=0; 
	END_IF
	
	i := i +1;
	IF (i >= MAX_CSV_ROWS)  THEN 
		i:=0; 
	END_IF
END_IF
	
// Verificações
//	Ao Deletar e salvar uma receita - O sistema deve verificar qual endereço ficou em vazio, e fazer uma rotina de reorganiza-lo e depois escrever na tabela de receitas
// Criar Receitar - verificar qual o ultima endereço da tabela vazia. Escrever ali o valores e ao apertar salvar escrever na tabela de receitas
//Editar e Cancelar - Não escreve na tabela

IF b_deletar_receita AND b_reorganizar = 0 THEN
	
	Recipe_Name_Select					:= '';
	Recipe_No_Select					:= 0;
	Recipe_ID_Select					:= 0;
		
	Recipe_Pontos_Solda_Select			:= 0;
		
	Recipe_P_X01_Solda_Select			:= 0.0;
	Recipe_P_Y01_Solda_Select			:= 0.0;
	Recipe_P01_Solda_Select				:= FALSE;
	Recipe_P_X02_Solda_Select			:= 0.0;
	Recipe_P_Y02_Solda_Select			:= 0.0;
	Recipe_P02_Solda_Select				:= FALSE;	
	Recipe_P_X03_Solda_Select			:= 0.0;
	Recipe_P_Y03_Solda_Select			:= 0.0;
	Recipe_P03_Solda_Select				:= FALSE;
	Recipe_P_X04_Solda_Select			:= 0.0;
	Recipe_P_Y04_Solda_Select			:= 0.0;
	Recipe_P04_Solda_Select				:= FALSE;
	Recipe_P_X05_Solda_Select			:= 0.0;
	Recipe_P_Y05_Solda_Select			:= 0.0;
	Recipe_P05_Solda_Select				:= FALSE;
	
	Recipe_P_X06_Solda_Select			:= 0.0;
	Recipe_P_Y06_Solda_Select			:= 0.0;
	Recipe_P06_Solda_Select				:= FALSE;
	Recipe_P_X07_Solda_Select			:= 0.0;
	Recipe_P_Y07_Solda_Select			:= 0.0;
	Recipe_P07_Solda_Select				:= FALSE;	
	Recipe_P_X08_Solda_Select			:= 0.0;
	Recipe_P_Y08_Solda_Select			:= 0.0;
	Recipe_P08_Solda_Select				:= FALSE;
	Recipe_P_X09_Solda_Select			:= 0.0;
	Recipe_P_Y09_Solda_Select			:= 0.0;
	Recipe_P09_Solda_Select				:= FALSE;
	Recipe_P_X10_Solda_Select			:= 0.0;
	Recipe_P_Y10_Solda_Select			:= 0.0;
	Recipe_P10_Solda_Select				:= FALSE;
		
	Recipe_P_X11_Solda_Select			:= 0.0;
	Recipe_P_Y11_Solda_Select			:= 0.0;
	Recipe_P11_Solda_Select				:= FALSE;
	Recipe_P_X12_Solda_Select			:= 0.0;
	Recipe_P_Y12_Solda_Select			:= 0.0;
	Recipe_P12_Solda_Select				:= FALSE;	
	Recipe_P_X13_Solda_Select			:= 0.0;
	Recipe_P_Y13_Solda_Select			:= 0.0;
	Recipe_P13_Solda_Select				:= FALSE;
	Recipe_P_X14_Solda_Select			:= 0.0;
	Recipe_P_Y14_Solda_Select			:= 0.0;
	Recipe_P14_Solda_Select				:= FALSE;
	Recipe_P_X15_Solda_Select			:= 0.0;
	Recipe_P_Y15_Solda_Select			:= 0.0;
	Recipe_P15_Solda_Select				:= FALSE;
		
	Recipe_Valvula_Proporcional_Select	:= 0.0;
	
	Recipe_Pontos_Camera_Select			:= 0;
	Recipe_JobID_F01_Camera_Select		:= 0;
	Recipe_JobID_F01_Camera_Select		:= 0;
	Recipe_JobID_F01_Camera_Select		:= 0;
	Recipe_JobID_F01_Camera_Select		:= 0;
	Recipe_JobID_F01_Camera_Select		:= 0;

	Recipe_Pecas_Caixa_Select			:= 0;
	
	IF b_cancelar_receita THEN
		
		b_deletar_receita := FALSE;
		b_cancelar_receita := FALSE;
		b_editar_receita := FALSE;
		
	ELSIF b_salvar_receita AND b_reorganizar = 0 THEN
		
		database_read[Recipe_select_int, 0] := '';
		database_read[Recipe_select_int, 1] := '';
		database_read[Recipe_select_int, 2] := '';
		database_read[Recipe_select_int, 3] := '';
		database_read[Recipe_select_int, 4] := '';
		database_read[Recipe_select_int, 5] := '';
		database_read[Recipe_select_int, 6] := '';
		database_read[Recipe_select_int, 7] := '';
		database_read[Recipe_select_int, 8] := '';
		database_read[Recipe_select_int, 9] := '';
		database_read[Recipe_select_int, 10] := '';
		database_read[Recipe_select_int, 11] := '';
		database_read[Recipe_select_int, 12] := '';
		database_read[Recipe_select_int, 13] := '';
		database_read[Recipe_select_int, 14] := '';
		database_read[Recipe_select_int, 15] := '';
		database_read[Recipe_select_int, 16] := '';
		database_read[Recipe_select_int, 17] := '';
		database_read[Recipe_select_int, 18] := '';
		database_read[Recipe_select_int, 19] := '';
		database_read[Recipe_select_int, 20] := '';
		database_read[Recipe_select_int, 21] := '';
		database_read[Recipe_select_int, 22] := '';
		database_read[Recipe_select_int, 23] := '';
		database_read[Recipe_select_int, 24] := '';
		database_read[Recipe_select_int, 25] := '';
		database_read[Recipe_select_int, 26] := '';
		database_read[Recipe_select_int, 27] := '';
		database_read[Recipe_select_int, 28] := '';
		database_read[Recipe_select_int, 29] := '';
		database_read[Recipe_select_int, 30] := '';
		database_read[Recipe_select_int, 31] := '';
		database_read[Recipe_select_int, 32] := '';
		database_read[Recipe_select_int, 33] := '';
		database_read[Recipe_select_int, 34] := '';
		database_read[Recipe_select_int, 35] := '';
		database_read[Recipe_select_int, 36] := '';
		database_read[Recipe_select_int, 37] := '';
		database_read[Recipe_select_int, 38] := '';
		database_read[Recipe_select_int, 39] := '';
		database_read[Recipe_select_int, 40] := '';
		database_read[Recipe_select_int, 41] := '';
		database_read[Recipe_select_int, 42] := '';
		database_read[Recipe_select_int, 43] := '';
		database_read[Recipe_select_int, 44] := '';
		database_read[Recipe_select_int, 45] := '';
		database_read[Recipe_select_int, 46] := '';
		database_read[Recipe_select_int, 47] := '';
		database_read[Recipe_select_int, 48] := '';
		database_read[Recipe_select_int, 49] := '';
		database_read[Recipe_select_int, 50] := '';
		database_read[Recipe_select_int, 51] := '';
		database_read[Recipe_select_int, 52] := '';
		database_read[Recipe_select_int, 53] := '';
		database_read[Recipe_select_int, 54] := '';
		database_read[Recipe_select_int, 55] := '';
		database_read[Recipe_select_int, 56] := '';
		Item_deletado := Recipe_select_int;
		b_reorganizar := 1;
		b_deletar_receita := FALSE;
		b_cancelar_receita := FALSE;
		b_editar_receita := FALSE;
		Simbolo_Atualizacao := TRUE;
		//Recipe_select_int := 0;
	END_IF

END_IF

IF b_reorganizar = 1 THEN
	Item_deletado := Item_deletado + 1;
	b_reorganizar := 2;
ELSIF b_reorganizar = 2 THEN
	
	Row_copy[0]		:= (database_read[Item_deletado, 0]);
	Row_copy[1]		:= (database_read[Item_deletado, 1]);
	Row_copy[2]		:= (database_read[Item_deletado, 2]);
	Row_copy[3]		:= (database_read[Item_deletado, 3]);
	Row_copy[4]		:= (database_read[Item_deletado, 4]);
	Row_copy[5]		:= (database_read[Item_deletado, 5]);
	Row_copy[6]		:= (database_read[Item_deletado, 6]);
	Row_copy[7]		:= (database_read[Item_deletado, 7]);
	Row_copy[8]		:= (database_read[Item_deletado, 8]);
	Row_copy[9]		:= (database_read[Item_deletado, 9]);
	Row_copy[10]	:= (database_read[Item_deletado, 10]);
	Row_copy[11]	:= (database_read[Item_deletado, 11]);
	Row_copy[12]	:= (database_read[Item_deletado, 12]);
	Row_copy[13]	:= (database_read[Item_deletado, 13]);
	Row_copy[14]	:= (database_read[Item_deletado, 14]);
	Row_copy[15]	:= (database_read[Item_deletado, 15]);
	Row_copy[16]	:= (database_read[Item_deletado, 16]);
	Row_copy[17]	:= (database_read[Item_deletado, 17]);
	Row_copy[18]	:= (database_read[Item_deletado, 18]);
	Row_copy[19]	:= (database_read[Item_deletado, 19]);
	Row_copy[20]	:= (database_read[Item_deletado, 20]);
	Row_copy[21]	:= (database_read[Item_deletado, 21]);
	Row_copy[22]	:= (database_read[Item_deletado, 22]);
	Row_copy[23]	:= (database_read[Item_deletado, 23]);
	Row_copy[24]	:= (database_read[Item_deletado, 24]);
	Row_copy[25]	:= (database_read[Item_deletado, 25]);
	Row_copy[26]	:= (database_read[Item_deletado, 26]);
	Row_copy[27]	:= (database_read[Item_deletado, 27]);
	Row_copy[28]	:= (database_read[Item_deletado, 28]);
	Row_copy[29]	:= (database_read[Item_deletado, 29]);
	Row_copy[30]	:= (database_read[Item_deletado, 30]);
	Row_copy[31]	:= (database_read[Item_deletado, 31]);
	Row_copy[32]	:= (database_read[Item_deletado, 32]);
	Row_copy[33]	:= (database_read[Item_deletado, 33]);
	Row_copy[34]	:= (database_read[Item_deletado, 34]);
	Row_copy[35]	:= (database_read[Item_deletado, 35]);
	Row_copy[36]	:= (database_read[Item_deletado, 36]);
	Row_copy[37]	:= (database_read[Item_deletado, 37]);
	Row_copy[38]	:= (database_read[Item_deletado, 38]);
	Row_copy[39]	:= (database_read[Item_deletado, 39]);
	Row_copy[40]	:= (database_read[Item_deletado, 40]);
	Row_copy[41]	:= (database_read[Item_deletado, 41]);
	Row_copy[42]	:= (database_read[Item_deletado, 42]);
	Row_copy[43]	:= (database_read[Item_deletado, 43]);
	Row_copy[44]	:= (database_read[Item_deletado, 44]);
	Row_copy[45]	:= (database_read[Item_deletado, 45]);
	Row_copy[46]	:= (database_read[Item_deletado, 46]);
	Row_copy[47]	:= (database_read[Item_deletado, 47]);
	Row_copy[48]	:= (database_read[Item_deletado, 48]);
	Row_copy[49]	:= (database_read[Item_deletado, 49]);
	Row_copy[50]	:= (database_read[Item_deletado, 50]);
	Row_copy[51]	:= (database_read[Item_deletado, 51]);
	Row_copy[52]	:= (database_read[Item_deletado, 52]);
	Row_copy[53]	:= (database_read[Item_deletado, 53]);
	Row_copy[54]	:= (database_read[Item_deletado, 54]);
	Row_copy[55]	:= (database_read[Item_deletado, 55]);
	Row_copy[56]	:= (database_read[Item_deletado, 56]);
	b_reorganizar := 3;

ELSIF b_reorganizar = 3 THEN
	
	database_read[(Item_deletado - 1), 0] := Row_copy[0];
	database_read[(Item_deletado - 1), 1] := Row_copy[1];
	database_read[(Item_deletado - 1), 2] := Row_copy[2];
	database_read[(Item_deletado - 1), 3] := Row_copy[3];
	database_read[(Item_deletado - 1), 4] := Row_copy[4];
	database_read[(Item_deletado - 1), 5] := Row_copy[5];
	database_read[(Item_deletado - 1), 6] := Row_copy[6];
	database_read[(Item_deletado - 1), 7] := Row_copy[7];
	database_read[(Item_deletado - 1), 8] := Row_copy[8];
	database_read[(Item_deletado - 1), 9] := Row_copy[9];
	database_read[(Item_deletado - 1), 10] := Row_copy[10];
	database_read[(Item_deletado - 1), 11] := Row_copy[11];
	database_read[(Item_deletado - 1), 12] := Row_copy[12];
	database_read[(Item_deletado - 1), 13] := Row_copy[13];
	database_read[(Item_deletado - 1), 14] := Row_copy[14];
	database_read[(Item_deletado - 1), 15] := Row_copy[15];
	database_read[(Item_deletado - 1), 16] := Row_copy[16];
	database_read[(Item_deletado - 1), 17] := Row_copy[17];
	database_read[(Item_deletado - 1), 18] := Row_copy[18];
	database_read[(Item_deletado - 1), 19] := Row_copy[19];
	database_read[(Item_deletado - 1), 20] := Row_copy[20];
	database_read[(Item_deletado - 1), 21] := Row_copy[21];
	database_read[(Item_deletado - 1), 22] := Row_copy[22];
	database_read[(Item_deletado - 1), 23] := Row_copy[23];
	database_read[(Item_deletado - 1), 24] := Row_copy[24];
	database_read[(Item_deletado - 1), 25] := Row_copy[25];
	database_read[(Item_deletado - 1), 26] := Row_copy[26];
	database_read[(Item_deletado - 1), 27] := Row_copy[27];
	database_read[(Item_deletado - 1), 28] := Row_copy[28];
	database_read[(Item_deletado - 1), 29] := Row_copy[29];
	database_read[(Item_deletado - 1), 30] := Row_copy[30];
	database_read[(Item_deletado - 1), 31] := Row_copy[31];
	database_read[(Item_deletado - 1), 32] := Row_copy[32];
	database_read[(Item_deletado - 1), 33] := Row_copy[33];
	database_read[(Item_deletado - 1), 34] := Row_copy[34];
	database_read[(Item_deletado - 1), 35] := Row_copy[35];
	database_read[(Item_deletado - 1), 36] := Row_copy[36];
	database_read[(Item_deletado - 1), 37] := Row_copy[37];
	database_read[(Item_deletado - 1), 38] := Row_copy[38];
	database_read[(Item_deletado - 1), 39] := Row_copy[39];
	database_read[(Item_deletado - 1), 40] := Row_copy[40];
	database_read[(Item_deletado - 1), 41] := Row_copy[41];
	database_read[(Item_deletado - 1), 42] := Row_copy[42];
	database_read[(Item_deletado - 1), 43] := Row_copy[43];
	database_read[(Item_deletado - 1), 44] := Row_copy[44];
	database_read[(Item_deletado - 1), 45] := Row_copy[45];
	database_read[(Item_deletado - 1), 46] := Row_copy[46];
	database_read[(Item_deletado - 1), 47] := Row_copy[47];
	database_read[(Item_deletado - 1), 48] := Row_copy[48];
	database_read[(Item_deletado - 1), 49] := Row_copy[49];
	database_read[(Item_deletado - 1), 50] := Row_copy[50];
	database_read[(Item_deletado - 1), 51] := Row_copy[51];
	database_read[(Item_deletado - 1), 52] := Row_copy[52];
	database_read[(Item_deletado - 1), 53] := Row_copy[53];
	database_read[(Item_deletado - 1), 54] := Row_copy[54];
	database_read[(Item_deletado - 1), 55] := Row_copy[55];
	database_read[(Item_deletado - 1), 56] := Row_copy[56];
	
	IF Item_deletado >= MAX_CSV_ROWS THEN
		Item_deletado := 0;
		b_reorganizar := 0;
		b_salvar_receita := FALSE;
		b_deletar_receita := FALSE;
		b_cancelar_receita := FALSE;
		b_editar_receita := FALSE;
		bWrite := TRUE;
		Recipe_select_int := 0;
	ELSE
		b_reorganizar := 1;	
	
	END_IF
END_IF
	
	
// Editar	
IF b_editar_receita AND NOT b_deletar_receita AND b_salvar_receita THEN
	
	database_read[Recipe_select_int, 0] := Recipe_Name_Select;
	database_read[Recipe_select_int, 1] := INT_TO_STRING (Recipe_No_Select);
	database_read[Recipe_select_int, 2] := INT_TO_STRING (Recipe_ID_Select);
	
	database_read[Recipe_select_int, 3] := INT_TO_STRING (Recipe_Pontos_Solda_Select);
	
	database_read[Recipe_select_int, 4] := LREAL_TO_STRING (Recipe_P_X01_Solda_Select);
	database_read[Recipe_select_int, 5] := LREAL_TO_STRING (Recipe_P_Y01_Solda_Select);
	database_read[Recipe_select_int, 6] := BOOL_TO_STRING (Recipe_P01_Solda_Select);
	database_read[Recipe_select_int, 7] := LREAL_TO_STRING (Recipe_P_X02_Solda_Select);
	database_read[Recipe_select_int, 8] := LREAL_TO_STRING (Recipe_P_Y02_Solda_Select);
	database_read[Recipe_select_int, 9] := BOOL_TO_STRING (Recipe_P02_Solda_Select);
	database_read[Recipe_select_int, 10] := LREAL_TO_STRING (Recipe_P_X03_Solda_Select);
	database_read[Recipe_select_int, 11] := LREAL_TO_STRING (Recipe_P_Y03_Solda_Select);
	database_read[Recipe_select_int, 12] := BOOL_TO_STRING (Recipe_P03_Solda_Select);
	database_read[Recipe_select_int, 13] := LREAL_TO_STRING (Recipe_P_X04_Solda_Select);
	database_read[Recipe_select_int, 14] := LREAL_TO_STRING (Recipe_P_Y04_Solda_Select);
	database_read[Recipe_select_int, 15] := BOOL_TO_STRING (Recipe_P04_Solda_Select);
	database_read[Recipe_select_int, 16] := LREAL_TO_STRING (Recipe_P_X05_Solda_Select);
	database_read[Recipe_select_int, 17] := LREAL_TO_STRING (Recipe_P_Y05_Solda_Select);
	database_read[Recipe_select_int, 18] := BOOL_TO_STRING (Recipe_P05_Solda_Select);
	
	database_read[Recipe_select_int, 19] := LREAL_TO_STRING (Recipe_P_X06_Solda_Select);
	database_read[Recipe_select_int, 20] := LREAL_TO_STRING (Recipe_P_Y06_Solda_Select);
	database_read[Recipe_select_int, 21] := BOOL_TO_STRING (Recipe_P06_Solda_Select);
	database_read[Recipe_select_int, 22] := LREAL_TO_STRING (Recipe_P_X07_Solda_Select);
	database_read[Recipe_select_int, 23] := LREAL_TO_STRING (Recipe_P_Y07_Solda_Select);
	database_read[Recipe_select_int, 24] := BOOL_TO_STRING (Recipe_P07_Solda_Select);
	database_read[Recipe_select_int, 25] := LREAL_TO_STRING (Recipe_P_X08_Solda_Select);
	database_read[Recipe_select_int, 26] := LREAL_TO_STRING (Recipe_P_Y08_Solda_Select);
	database_read[Recipe_select_int, 27] := BOOL_TO_STRING (Recipe_P08_Solda_Select);
	database_read[Recipe_select_int, 28] := LREAL_TO_STRING (Recipe_P_X09_Solda_Select);
	database_read[Recipe_select_int, 29] := LREAL_TO_STRING (Recipe_P_Y09_Solda_Select);
	database_read[Recipe_select_int, 30] := BOOL_TO_STRING (Recipe_P09_Solda_Select);
	database_read[Recipe_select_int, 31] := LREAL_TO_STRING (Recipe_P_X10_Solda_Select);
	database_read[Recipe_select_int, 32] := LREAL_TO_STRING (Recipe_P_Y10_Solda_Select);
	database_read[Recipe_select_int, 33] := BOOL_TO_STRING (Recipe_P10_Solda_Select);
	
	database_read[Recipe_select_int, 34] := LREAL_TO_STRING (Recipe_P_X11_Solda_Select);
	database_read[Recipe_select_int, 35] := LREAL_TO_STRING (Recipe_P_Y11_Solda_Select);
	database_read[Recipe_select_int, 36] := BOOL_TO_STRING (Recipe_P11_Solda_Select);
	database_read[Recipe_select_int, 37] := LREAL_TO_STRING (Recipe_P_X12_Solda_Select);
	database_read[Recipe_select_int, 38] := LREAL_TO_STRING (Recipe_P_Y12_Solda_Select);
	database_read[Recipe_select_int, 39] := BOOL_TO_STRING (Recipe_P12_Solda_Select);
	database_read[Recipe_select_int, 40] := LREAL_TO_STRING (Recipe_P_X13_Solda_Select);
	database_read[Recipe_select_int, 41] := LREAL_TO_STRING (Recipe_P_Y13_Solda_Select);
	database_read[Recipe_select_int, 42] := BOOL_TO_STRING (Recipe_P13_Solda_Select);
	database_read[Recipe_select_int, 43] := LREAL_TO_STRING (Recipe_P_X14_Solda_Select);
	database_read[Recipe_select_int, 44] := LREAL_TO_STRING (Recipe_P_Y14_Solda_Select);
	database_read[Recipe_select_int, 45] := BOOL_TO_STRING (Recipe_P14_Solda_Select);
	database_read[Recipe_select_int, 46] := LREAL_TO_STRING (Recipe_P_X15_Solda_Select);
	database_read[Recipe_select_int, 47] := LREAL_TO_STRING (Recipe_P_Y15_Solda_Select);
	database_read[Recipe_select_int, 48] := BOOL_TO_STRING (Recipe_P15_Solda_Select);
	
	database_read[Recipe_select_int, 49] := LREAL_TO_STRING (Recipe_Valvula_Proporcional_Select);
	
	database_read[Recipe_select_int, 50] := INT_TO_STRING (Recipe_Pontos_Camera_Select);
	database_read[Recipe_select_int, 51] := INT_TO_STRING (Recipe_JobID_F01_Camera_Select);
	database_read[Recipe_select_int, 52] := INT_TO_STRING (Recipe_JobID_F02_Camera_Select);
	database_read[Recipe_select_int, 53] := INT_TO_STRING (Recipe_JobID_F03_Camera_Select);
	database_read[Recipe_select_int, 54] := INT_TO_STRING (Recipe_JobID_F04_Camera_Select);
	database_read[Recipe_select_int, 55] := INT_TO_STRING (Recipe_JobID_F05_Camera_Select);
	
	database_read[Recipe_select_int, 56] := INT_TO_STRING (Recipe_Pecas_Caixa_Select);
	
	b_salvar_receita := FALSE;
	b_editar_receita := FALSE;
	bWrite := TRUE;
	
ELSIF	
	b_editar_receita AND NOT b_deletar_receita AND b_cancelar_receita THEN
	b_cancelar_receita := FALSE;
	b_editar_receita := FALSE;
	
END_IF

// Criar nova receita
IF b_criar_receita THEN
	
	CASE PassoLimparMemoriasReceita OF
		
		0: //Limpar Memórias "Recipe" da Receita
			
			Recipe_Name_Select					:= '';
			Recipe_No_Select					:= 0;
			Recipe_ID_Select					:= 0;
				
			Recipe_Pontos_Solda_Select			:= 0;
				
			Recipe_P_X01_Solda_Select			:= 0.0;
			Recipe_P_Y01_Solda_Select			:= 0.0;
			Recipe_P01_Solda_Select				:= FALSE;
			Recipe_P_X02_Solda_Select			:= 0.0;
			Recipe_P_Y02_Solda_Select			:= 0.0;
			Recipe_P02_Solda_Select				:= FALSE;	
			Recipe_P_X03_Solda_Select			:= 0.0;
			Recipe_P_Y03_Solda_Select			:= 0.0;
			Recipe_P03_Solda_Select				:= FALSE;
			Recipe_P_X04_Solda_Select			:= 0.0;
			Recipe_P_Y04_Solda_Select			:= 0.0;
			Recipe_P04_Solda_Select				:= FALSE;
			Recipe_P_X05_Solda_Select			:= 0.0;
			Recipe_P_Y05_Solda_Select			:= 0.0;
			Recipe_P05_Solda_Select				:= FALSE;
			
			Recipe_P_X06_Solda_Select			:= 0.0;
			Recipe_P_Y06_Solda_Select			:= 0.0;
			Recipe_P06_Solda_Select				:= FALSE;
			Recipe_P_X07_Solda_Select			:= 0.0;
			Recipe_P_Y07_Solda_Select			:= 0.0;
			Recipe_P07_Solda_Select				:= FALSE;	
			Recipe_P_X08_Solda_Select			:= 0.0;
			Recipe_P_Y08_Solda_Select			:= 0.0;
			Recipe_P08_Solda_Select				:= FALSE;
			Recipe_P_X09_Solda_Select			:= 0.0;
			Recipe_P_Y09_Solda_Select			:= 0.0;
			Recipe_P09_Solda_Select				:= FALSE;
			Recipe_P_X10_Solda_Select			:= 0.0;
			Recipe_P_Y10_Solda_Select			:= 0.0;
			Recipe_P10_Solda_Select				:= FALSE;
				
			Recipe_P_X11_Solda_Select			:= 0.0;
			Recipe_P_Y11_Solda_Select			:= 0.0;
			Recipe_P11_Solda_Select				:= FALSE;
			Recipe_P_X12_Solda_Select			:= 0.0;
			Recipe_P_Y12_Solda_Select			:= 0.0;
			Recipe_P12_Solda_Select				:= FALSE;	
			Recipe_P_X13_Solda_Select			:= 0.0;
			Recipe_P_Y13_Solda_Select			:= 0.0;
			Recipe_P13_Solda_Select				:= FALSE;
			Recipe_P_X14_Solda_Select			:= 0.0;
			Recipe_P_Y14_Solda_Select			:= 0.0;
			Recipe_P14_Solda_Select				:= FALSE;
			Recipe_P_X15_Solda_Select			:= 0.0;
			Recipe_P_Y15_Solda_Select			:= 0.0;
			Recipe_P15_Solda_Select				:= FALSE;
				
			Recipe_Valvula_Proporcional_Select	:= 0.0;
			
			Recipe_Pontos_Camera_Select			:= 0;
			Recipe_JobID_F01_Camera_Select		:= 0;
			Recipe_JobID_F01_Camera_Select		:= 0;
			Recipe_JobID_F01_Camera_Select		:= 0;
			Recipe_JobID_F01_Camera_Select		:= 0;
			Recipe_JobID_F01_Camera_Select		:= 0;
		
			Recipe_Pecas_Caixa_Select			:= 0;
			
			PassoLimparMemoriasReceita := 10;
	
	END_CASE

ELSE
	
	PassoLimparMemoriasReceita := 0;	

END_IF

IF b_criar_receita AND b_salvar_receita THEN
	
	database_read[Item_livre, 0] := Recipe_Name_Select;
	database_read[Item_livre, 1] := INT_TO_STRING (Recipe_No_Select);
	database_read[Item_livre, 2] := INT_TO_STRING (Recipe_ID_Select);
	
	database_read[Item_livre, 3] := INT_TO_STRING (Recipe_Pontos_Solda_Select);
	
	database_read[Item_livre, 4] := LREAL_TO_STRING (Recipe_P_X01_Solda_Select);
	database_read[Item_livre, 5] := LREAL_TO_STRING (Recipe_P_Y01_Solda_Select);
	database_read[Item_livre, 6] := BOOL_TO_STRING (Recipe_P01_Solda_Select);
	database_read[Item_livre, 7] := LREAL_TO_STRING (Recipe_P_X02_Solda_Select);
	database_read[Item_livre, 8] := LREAL_TO_STRING (Recipe_P_Y02_Solda_Select);
	database_read[Item_livre, 9] := BOOL_TO_STRING (Recipe_P02_Solda_Select);
	database_read[Item_livre, 10] := LREAL_TO_STRING (Recipe_P_X03_Solda_Select);
	database_read[Item_livre, 11] := LREAL_TO_STRING (Recipe_P_Y03_Solda_Select);
	database_read[Item_livre, 12] := BOOL_TO_STRING (Recipe_P03_Solda_Select);
	database_read[Item_livre, 13] := LREAL_TO_STRING (Recipe_P_X04_Solda_Select);
	database_read[Item_livre, 14] := LREAL_TO_STRING (Recipe_P_Y04_Solda_Select);
	database_read[Item_livre, 15] := BOOL_TO_STRING (Recipe_P04_Solda_Select);
	database_read[Item_livre, 16] := LREAL_TO_STRING (Recipe_P_X05_Solda_Select);
	database_read[Item_livre, 17] := LREAL_TO_STRING (Recipe_P_Y05_Solda_Select);
	database_read[Item_livre, 18] := BOOL_TO_STRING (Recipe_P05_Solda_Select);
	
	database_read[Item_livre, 19] := LREAL_TO_STRING (Recipe_P_X06_Solda_Select);
	database_read[Item_livre, 20] := LREAL_TO_STRING (Recipe_P_Y06_Solda_Select);
	database_read[Item_livre, 21] := BOOL_TO_STRING (Recipe_P06_Solda_Select);
	database_read[Item_livre, 22] := LREAL_TO_STRING (Recipe_P_X07_Solda_Select);
	database_read[Item_livre, 23] := LREAL_TO_STRING (Recipe_P_Y07_Solda_Select);
	database_read[Item_livre, 24] := BOOL_TO_STRING (Recipe_P07_Solda_Select);
	database_read[Item_livre, 25] := LREAL_TO_STRING (Recipe_P_X08_Solda_Select);
	database_read[Item_livre, 26] := LREAL_TO_STRING (Recipe_P_Y08_Solda_Select);
	database_read[Item_livre, 27] := BOOL_TO_STRING (Recipe_P08_Solda_Select);
	database_read[Item_livre, 28] := LREAL_TO_STRING (Recipe_P_X09_Solda_Select);
	database_read[Item_livre, 29] := LREAL_TO_STRING (Recipe_P_Y09_Solda_Select);
	database_read[Item_livre, 30] := BOOL_TO_STRING (Recipe_P09_Solda_Select);
	database_read[Item_livre, 31] := LREAL_TO_STRING (Recipe_P_X10_Solda_Select);
	database_read[Item_livre, 32] := LREAL_TO_STRING (Recipe_P_Y10_Solda_Select);
	database_read[Item_livre, 33] := BOOL_TO_STRING (Recipe_P10_Solda_Select);
	
	database_read[Item_livre, 34] := LREAL_TO_STRING (Recipe_P_X11_Solda_Select);
	database_read[Item_livre, 35] := LREAL_TO_STRING (Recipe_P_Y11_Solda_Select);
	database_read[Item_livre, 36] := BOOL_TO_STRING (Recipe_P11_Solda_Select);
	database_read[Item_livre, 37] := LREAL_TO_STRING (Recipe_P_X12_Solda_Select);
	database_read[Item_livre, 38] := LREAL_TO_STRING (Recipe_P_Y12_Solda_Select);
	database_read[Item_livre, 39] := BOOL_TO_STRING (Recipe_P12_Solda_Select);
	database_read[Item_livre, 40] := LREAL_TO_STRING (Recipe_P_X13_Solda_Select);
	database_read[Item_livre, 41] := LREAL_TO_STRING (Recipe_P_Y13_Solda_Select);
	database_read[Item_livre, 42] := BOOL_TO_STRING (Recipe_P13_Solda_Select);
	database_read[Item_livre, 43] := LREAL_TO_STRING (Recipe_P_X14_Solda_Select);
	database_read[Item_livre, 44] := LREAL_TO_STRING (Recipe_P_Y14_Solda_Select);
	database_read[Item_livre, 45] := BOOL_TO_STRING (Recipe_P14_Solda_Select);
	database_read[Item_livre, 46] := LREAL_TO_STRING (Recipe_P_X15_Solda_Select);
	database_read[Item_livre, 47] := LREAL_TO_STRING (Recipe_P_Y15_Solda_Select);
	database_read[Item_livre, 48] := BOOL_TO_STRING (Recipe_P15_Solda_Select);
	
	database_read[Item_livre, 49] := LREAL_TO_STRING (Recipe_Valvula_Proporcional_Select);
	
	database_read[Item_livre, 50] := INT_TO_STRING (Recipe_Pontos_Camera_Select);
	database_read[Item_livre, 51] := INT_TO_STRING (Recipe_JobID_F01_Camera_Select);
	database_read[Item_livre, 52] := INT_TO_STRING (Recipe_JobID_F02_Camera_Select);
	database_read[Item_livre, 53] := INT_TO_STRING (Recipe_JobID_F03_Camera_Select);
	database_read[Item_livre, 54] := INT_TO_STRING (Recipe_JobID_F04_Camera_Select);
	database_read[Item_livre, 55] := INT_TO_STRING (Recipe_JobID_F05_Camera_Select);
	
	database_read[Item_livre, 56] := INT_TO_STRING (Recipe_Pecas_Caixa_Select);

	b_salvar_receita := FALSE;
	b_criar_receita := FALSE;
	bWrite := TRUE;

ELSIF 	b_criar_receita AND b_cancelar_receita THEN
	b_criar_receita := FALSE;
	b_cancelar_receita := FALSE;
	
END_IF

(*===================		EXECUTAR RECEITA		======================*)

IF b_executar_receita THEN
	
	// := Recipe_Name_Select;
	// := Recipe_No_Select;
	// := Recipe_ID_Select;
	
	NumPontosSolda := Recipe_Pontos_Solda_Select;
	
	TargetX[0] := Recipe_P_X01_Solda_Select;
	TargetY[0] := Recipe_P_Y01_Solda_Select;
	SoldaXY[0] := Recipe_P01_Solda_Select;
	TargetX[1] := Recipe_P_X02_Solda_Select;
	TargetY[1] := Recipe_P_Y02_Solda_Select;
	SoldaXY[1] := Recipe_P02_Solda_Select;
	TargetX[2] := Recipe_P_X03_Solda_Select;
	TargetY[2] := Recipe_P_Y03_Solda_Select;
	SoldaXY[2] := Recipe_P03_Solda_Select;
	TargetX[3] := Recipe_P_X04_Solda_Select;
	TargetY[3] := Recipe_P_Y04_Solda_Select;
	SoldaXY[3] := Recipe_P04_Solda_Select;
	TargetX[4] := Recipe_P_X05_Solda_Select;
	TargetY[4] := Recipe_P_Y05_Solda_Select;
	SoldaXY[4] := Recipe_P05_Solda_Select;
	
	TargetX[5] := Recipe_P_X06_Solda_Select;
	TargetY[5] := Recipe_P_Y06_Solda_Select;
	SoldaXY[5] := Recipe_P06_Solda_Select;
	TargetX[6] := Recipe_P_X07_Solda_Select;
	TargetY[6] := Recipe_P_Y07_Solda_Select;
	SoldaXY[6] := Recipe_P07_Solda_Select;
	TargetX[7] := Recipe_P_X08_Solda_Select;
	TargetY[7] := Recipe_P_Y08_Solda_Select;
	SoldaXY[7] := Recipe_P08_Solda_Select;
	TargetX[8] := Recipe_P_X09_Solda_Select;
	TargetY[8] := Recipe_P_Y09_Solda_Select;
	SoldaXY[8] := Recipe_P09_Solda_Select;
	TargetX[9] := Recipe_P_X10_Solda_Select;
	TargetY[9] := Recipe_P_Y10_Solda_Select;
	SoldaXY[9] := Recipe_P10_Solda_Select;
	
	TargetX[10] := Recipe_P_X11_Solda_Select;
	TargetY[10] := Recipe_P_Y11_Solda_Select;
	SoldaXY[10] := Recipe_P11_Solda_Select;
	TargetX[11] := Recipe_P_X12_Solda_Select;
	TargetY[11] := Recipe_P_Y12_Solda_Select;
	SoldaXY[11] := Recipe_P12_Solda_Select;
	TargetX[12] := Recipe_P_X13_Solda_Select;
	TargetY[12] := Recipe_P_Y13_Solda_Select;
	SoldaXY[12] := Recipe_P13_Solda_Select;
	TargetX[13] := Recipe_P_X14_Solda_Select;
	TargetY[13] := Recipe_P_Y14_Solda_Select;
	SoldaXY[13] := Recipe_P14_Solda_Select;
	TargetX[14] := Recipe_P_X15_Solda_Select;
	TargetY[14] := Recipe_P_Y15_Solda_Select;
	SoldaXY[14] := Recipe_P15_Solda_Select;
		
	// := Recipe_Valvula_Proporcional_Select;
	
	// := Recipe_Pontos_Camera_Select;
	CameraJobID[0] := Recipe_JobID_F01_Camera_Select;
	CameraJobID[1] := Recipe_JobID_F02_Camera_Select;
	CameraJobID[2] := Recipe_JobID_F03_Camera_Select;
	CameraJobID[3] := Recipe_JobID_F04_Camera_Select;
	CameraJobID[4] := Recipe_JobID_F05_Camera_Select;
	
	// := Recipe_Pecas_Caixa_Select;
	
	b_executar_receita := FALSE;
//	ServoTest := TRUE;
	
END_IF

(*========================================================================*)

END_PROGRAM

// ---- POUs/Receita/P_Read_Tabela.TcPOU
PROGRAM P_Read_Tabela
(* Reading of CSV file in text mode. None of the field value is containing any non-printing control characters like line feed, carriage return, quotation marks, semicolon... *)
VAR
//	bRead			: BOOL := FALSE;(* Rising edge starts program execution *)
	sNetId			: T_AmsNetId := '';	(* TwinCAT system network address *)
	sFileName		: T_MaxString := 'C:\Users\User\Desktop\PLC\Softwares de Máquinas\Indab\Receitas\Receitas_Carrossel.csv';(* CSV destination file path and name *)
	//sFileName		: T_MaxString := '\Hard Disk\Receitas\Receitas_Carrossel.csv';(* CSV destination file path and name *)
	//sFileName		: T_MaxString := 'C:\Users\User\Desktop\PLC\Softwares de Máquinas\Indab\Receitas\Receitas_Carrossel.csv';(* CSV destination file path and name *)
	//sCSVLine		: T_MaxString := '';(* Single CSV text line (row, record), we are using string as record buffer (your are able to see read fields)  *)
	sCSVLine		: STRING (3000);
	sCSVField		: T_MaxString := '';(* Single CSV field value (column, record field) *)
	bBusy			: BOOL;
	bError			: BOOL;
	nErrId			: UDINT;
	nRow	 		: UDINT 	:= 0;(* Row number (record) *)
	nColumn			: UDINT 	:= 0;(* Column number (record field) *)
	hFile			: UINT		:= 0;(* File handle of the source file *)
	step			: DWORD 	:= 0;
	fbFileOpen		: FB_FileOpen;(* Opens file *)
	fbFileClose		: FB_FileClose;(* Closes file *)
	fbFileGets		: FB_FileGets;(* Reads one record (line) *)
	fbReader		: FB_CSVMemBufferReader;(* Helper function block used to parse CSV data bytes (single record line) *)

//	database		: ARRAY[0..MAX_CSV_ROWS, 0..MAX_CSV_COLUMNS ] OF STRING(MAX_CSV_FIELD_LENGTH);(* Target PLC database *)
END_VAR

CASE step OF
	0:	(* Wait for rising edge at bRead variable *)
		IF bRead THEN
			bRead 		:= FALSE;
			bBusy 		:= TRUE;
			bError		:= FALSE;
			nErrId		:= 0;
			hFile		:= 0;
			nRow	 	:= 0;
			nColumn		:= 0;
			MEMSET( ADR( database_read ), 0, SIZEOF( database_read ) );
			Simbolo_Atualizacao := TRUE;
			step 		:= 1;
		END_IF

	1:	(* Open source file *)
		fbFileOpen(  bExecute := FALSE  );
		fbFileOpen(  sNetId := sNetId, sPathName := sFileName, nMode := FOPEN_MODEREAD OR FOPEN_MODETEXT,(* Open file in TEXT mode! *)
					 ePath := PATH_GENERIC, bExecute := TRUE );
		step := 2;

	2:(* Wait until open not busy *)
		fbFileOpen( bExecute := FALSE, bError => bError, nErrID => nErrID, hFile => hFile );
		IF NOT fbFileOpen.bBusy THEN
			IF NOT fbFileOpen.bError THEN
				step := 3;
			ELSE(* Error: file not found? *)
				step := 100;
			END_IF
		END_IF

	3:	(* Read single line (record) *)
		fbFileGets( bExecute := FALSE );
		fbFileGets( sNetId := sNetId, hFile := hFile, bExecute := TRUE );
		step := 4;

	4:(* Wait until read not busy *)
		fbFileGets( bExecute := FALSE, bError => bError, nErrID => nErrID, sLine => sCSVLine );
		IF NOT fbFileGets.bBusy THEN
			IF NOT fbFileGets.bError THEN
				IF fbFileGets.bEOF THEN
					step := 10;(* End of file reached => Close source file *)
				ELSE

					(* FB_FileGets returns text line without the CR (carriage return) character.
					We have to restore the CR character (replace the $L character with $R$L characters) *)
					IF RIGHT( sCSVLine, 1 ) = '$L' THEN
						sCSVLine := REPLACE( sCSVLine, '$R$L', 2, LEN( sCSVLine ) );
					END_IF

					step := 5;
				END_IF
			ELSE(* Error *)
				step := 100;
			END_IF
		END_IF

	5:(* Parse single line (record) *)
		fbReader.eCmd := eEnumCmd_First;(* Read first field value *)
		REPEAT
			fbReader( pBuffer := ADR( sCSVLine ), cbBuffer := SIZEOF( sCSVLine ), getValue =>sCSVField );
			IF fbReader.bOk THEN
				fbReader.eCmd := eEnumCmd_Next;(* Read next field value *)

				IF ( nRow <= MAX_CSV_ROWS ) THEN
					IF ( nColumn <= MAX_CSV_COLUMNS ) THEN
						database_read[nRow, nColumn] := CSVFIELD_TO_STRING( sCSVField, FALSE );(* TODO: Save or use the field value in your application *)
					END_IF
				END_IF

				nColumn := nColumn + 1;(* Increment number of read columns *)
				IF fbReader.bCRLF THEN(* CRLF == TRUE => End of reacord reached *)
					nRow 		:= nRow + 1;(* Increment number of read records *)
					nColumn 	:= 0;(* Reset number of columns *)
				END_IF

			ELSE(* Error: End of record reached or all fields read *)
				step := 3;(* Try to read next line *)
			END_IF
		UNTIL NOT fbReader.bOk
		END_REPEAT

	10:	(* Close source file *)
		fbFileClose( bExecute := FALSE );
		fbFileClose( sNetId := sNetId, hFile := hFile, bExecute := TRUE );
		step := 11;

	11:(* Wait until close not busy *)
		fbFileClose( bExecute := FALSE, bError => bError, nErrID => nErrID );
		IF ( NOT fbFileClose.bBusy ) THEN
			hFile := 0;
			step := 100;
		END_IF

	100: (* Error or ready step => cleanup *)
		IF ( hFile <> 0 ) THEN
			step := 10; (* Close the source file *)
		ELSE
			bBusy := FALSE;
			step := 0;	(* Ready *)
			Simbolo_Atualizacao := FALSE;
		END_IF

END_CASE

END_PROGRAM

// ---- POUs/Receita/P_Write_Tabela.TcPOU
PROGRAM P_Write_Tabela
(* Writing of CSV file in text mode. None of the field value is containing any non-printing control characters like line feed, carriage return, quotation marks, semicolon... *)
VAR
//	bWrite			: BOOL := FALSE;(* Rising edge starts program execution *)
	sNetId			: T_AmsNetId := '';	(* TwinCAT system network address *)
	sFileName		: T_MaxString := 'C:\Users\User\Desktop\PLC\Softwares de Máquinas\Indab\Receitas\Receitas_Carrossel.csv';(* CSV destination file path and name *)
	//sFileName		: T_MaxString := '\Hard Disk\Receitas\Receitas_Carrossel.csv';(* CSV destination file path and name *)
	//sFileName		: T_MaxString := 'C:\Users\User\Desktop\PLC\Softwares de Máquinas\Indab\Receitas\Receitas_Carrossel.csv';(* CSV destination file path and name *)	
	sCSVLine		: T_MaxString := '';(* Single CSV text line (row, record), we are using string as record buffer (your are able to see created fields) *)
	sCSVField		: T_MaxString := '';(* Single CSV field value (column, record field) *)
	bBusy			: BOOL;
	bError			: BOOL;
	nErrId			: UDINT;
	nRow	 		: UDINT 	:= 0;(* Row number (record) *)
	nColumn			: UDINT 	:= 0;(* Column number (record field) *)
	hFile			: UINT		:= 0;(* File handle of the source file *)
	step			: DWORD 	:= 0;
	fbFileOpen		: FB_FileOpen;(* Opens file *)
	fbFileClose		: FB_FileClose;(* Closes file *)
	fbFilePuts		: FB_FilePuts;(* Writes one record (line) *)
	fbWriter		: FB_CSVMemBufferWriter;(* Helper function block used to create CSV data bytes (single record line) *)

	database		: ARRAY[0..MAX_CSV_ROWS, 0..MAX_CSV_COLUMNS ] OF STRING(MAX_CSV_FIELD_LENGTH);
	
	string_escrita	: T_MaxString;
	
	TON_ESCRITA		: TON;
	
END_VAR

database := database_read;

CASE step OF
	0:	(* Wait for rising edge at bWrite variable *)
		IF bWrite THEN
			bWrite 		:= FALSE;
			bBusy 		:= TRUE;
			bError		:= FALSE;
			nErrId		:= 0;
			hFile		:= 0;
			nRow	 	:= 0;
			nColumn		:= 0;
			step 		:= 1;
			Simbolo_Atualizacao := TRUE;
			TON_ESCRITA (IN:= TRUE);
		END_IF

	1:	(* Open source file *)
		fbFileOpen(  bExecute := FALSE  );
		fbFileOpen( 	sNetId := sNetId, sPathName := sFileName, nMode := FOPEN_MODEWRITE OR FOPEN_MODETEXT,(* Open file in TEXT mode! *)
						ePath := PATH_GENERIC, bExecute := TRUE );
		step := 2;

	2:(* Wait until open not busy *)
		fbFileOpen( bExecute := FALSE, bError => bError, nErrID => nErrID, hFile => hFile );
		IF NOT fbFileOpen.bBusy THEN
			IF NOT fbFileOpen.bError THEN
				step := 30;
			ELSE(* Error: file not found? *)
				step := 200;
			END_IF
		END_IF
		
		
	30:
			
		string_escrita := '';
		fbWriter.eCmd := eEnumCmd_First;(* Write first field value *)
		IF nRow <= (Main_Receita.Item_livre + 2)(*MAX_CSV_ROWS*) THEN

			IF nColumn < MAX_CSV_COLUMNS THEN
				
				string_escrita := database[ nRow, nColumn ];
				
				
				string_escrita := CONCAT (STR1 := string_escrita, STR2 := ';');
				(* Add new field to the record buffer 
				fbWriter( 	pBuffer := ADR( string_escrita ), cbBuffer := SIZEOF( string_escrita ) - 1, putValue := sCSVField, pValue := 0, cbValue := 0,
							bCRLF := ( nColumn = MAX_CSV_COLUMNS ) );(* bCRLF == TRUE => Write CRLF after the last field value *)
				IF fbWriter.bOk THEN
					fbWriter.eCmd := eEnumCmd_Next; Write next field value *)
					nColumn := nColumn + 1;
					step := 40;
			//	ELSE(* Error *)
			//		step := 100;
			//		RETURN;
			//	END_IF
			
			ELSE
				nColumn := 0;
				step := 33;	
			
			END_IF
		
		ELSE(* All rows written => Close file *)
			step := 100;
		END_IF	
			
		

	33:(* Convert one PLC record to CSV format *)
		
		string_escrita := 'ACABOU;$0A';
			(* FB_FilePuts adds allready CR (carriage return) to the written line.
			We have to replace the $R$L characters with $L character to avoid double CR. *)
		IF RIGHT( string_escrita, 2 ) = '$R$L' THEN
			string_escrita := REPLACE( string_escrita, '$L', 2, LEN( string_escrita ) - 1 );
		END_IF

		nRow := nRow + 1;(* Increment number of created records (rows) *)
		step := 40;(* Write record to the file *)

		

	40:	(* Write single text line *)
		
		fbFilePuts( bExecute := FALSE );
		fbFilePuts( sNetId := sNetId, hFile := hFile, sLine := string_escrita, bExecute := TRUE );
		step := 50;

	50:(* Wait until write not busy *)
		fbFilePuts( bExecute := FALSE, bError => bError, nErrID => nErrID );
		IF NOT fbFilePuts.bBusy THEN
			IF NOT fbFilePuts.bError THEN
				IF nColumn = 0 AND nRow >= MAX_CSV_ROWS THEN
					step := 100;(* Write next record *)
				ELSE 
					step := 30;	
				END_IF	
			ELSE(* Error *)
				step := 100;
			END_IF
		END_IF
		

	100:	(* Close source file *)
		fbFileClose( bExecute := FALSE );
		fbFileClose( sNetId := sNetId, hFile := hFile, bExecute := TRUE );
		step := 110;

	110:(* Wait until close not busy *)
		fbFileClose( bExecute := FALSE, bError => bError, nErrID => nErrID );
		IF ( NOT fbFileClose.bBusy ) THEN
			hFile := 0;
			step := 200;
		END_IF

	200: (* Error or ready step => cleanup *)
		IF ( hFile <> 0 ) THEN
			step := 100; (* Close the source file *)
		ELSE
			bBusy := FALSE;
			step := 0;	(* Ready *)
			Simbolo_Atualizacao := FALSE;
			bRead := TRUE;
		END_IF

END_CASE

TON_ESCRITA (pt := T#120S);

END_PROGRAM

// ---- POUs/CondicoesIniciais.TcPOU
PROGRAM CondicoesIniciais
VAR
		
	PassoCondicoesIniciais			: INT;
	
	EixoX_MoveAbsoluteOrigem		: MC_MoveAbsolute;
	EixoY_MoveAbsoluteOrigem		: MC_MoveAbsolute;
	
	Flag_EixoX_PosicaoOK			: BOOL;
	Flag_EixoY_PosicaoOK			: BOOL;
	
	DelayTest						: TON;
	
END_VAR

(*=====================		CONDIÇÕES INICIAIS		======================*)	

//Condição de Bloqueio da Máquina de Estados - Mesa Index FWD
IF (Alarmes.AlarmeGrave
	OR MaquinaLigada
	OR MaquinaModoManual
	OR NOT IhmBt_CondIniciais
	) THEN
	PassoCondicoesIniciais := 1000;
	EixoX_MoveAbsoluteOrigem(	Axis:= EixoX, Execute:= FALSE);
	EixoY_MoveAbsoluteOrigem(	Axis:= EixoY, Execute:= FALSE);
	Flag_EixoX_PosicaoOK := FALSE;
	Flag_EixoY_PosicaoOK := FALSE;

END_IF
CASE PassoCondicoesIniciais OF

	//Passo 0 - Inicialização
	0: PassoCondicoesIniciais := 10;
	
	//Passo 10 - Condição para iniciar Rotina de Condições Iniciais
	10: IF (IhmBt_CondIniciais) THEN
			PassoCondicoesIniciais := 20;
		END_IF
		
	//Passo 20 - Recuar Cilindro Principal
	20: LigarValvulaY6:= FALSE;
		LigarValvulaY9 := FALSE;
	IF (ReguaPotenciometricaSinal > 500 AND ReguaPotenciometricaSinal < 15000) THEN
		DelayTest(IN := TRUE, PT := T#5S);
		IF (DelayTest.Q) THEN
			PassoCondicoesIniciais := 30;
		END_IF
	END_IF

	//Passo 30 - Posicionar Servos X e Y - Ponto Inicial de Soldagem
	30: EixoX_MoveAbsoluteOrigem(	Axis := EixoX, 
									Execute := TRUE,
									Position := PosicaoOrigemX,
									Velocity := 1000
									//Acceleration:= 15000,
									//Deceleration:= 15000
									);
		IF (EixoX_MoveAbsoluteOrigem.Done) THEN
			Flag_EixoX_PosicaoOK := TRUE;	
		END_IF
		
		EixoY_MoveAbsoluteOrigem(	Axis := EixoY, 
									Execute := TRUE,
									Position := PosicaoOrigemY,
									Velocity := 1000
									//Acceleration:= 15000,
									//Deceleration:= 15000
									);
		IF (EixoY_MoveAbsoluteOrigem.Done) THEN
			Flag_EixoY_PosicaoOK := TRUE;	
		END_IF
		
		IF (Flag_EixoX_PosicaoOK AND Flag_EixoY_PosicaoOK) THEN
			PassoCondicoesIniciais := 40;	
		END_IF
		
	//Passo 40 - Finalizar Movimentação - Servos X e Y
	40: EixoX_MoveAbsoluteOrigem(	Axis:= EixoX, Execute:= FALSE);
		EixoY_MoveAbsoluteOrigem(	Axis:= EixoY, Execute:= FALSE);
		Flag_EixoX_PosicaoOK := FALSE;
		Flag_EixoY_PosicaoOK := FALSE;
		IhmBt_CondIniciais := FALSE;
		PassoCondicoesIniciais := 1000;
	
	//Passo 1000 - Finalização
	1000: 	IhmBt_CondIniciais := FALSE;
			PassoCondicoesIniciais := 0;
			

END_CASE

(*CASE PassoCondicoesIniciais OF

	//Passo 0 - Inicialização
	0: PassoCondicoesIniciais := 10;
	
	//Passo 10 - Condição para iniciar Rotina de Condições Iniciais
	10: //IF InComandoPedal THEN
			PassoCondicoesIniciais := 30;
		//END_IF
	
	//Passo 20 - Máquina de Solda em Condições Iniciais
	20:	
		PassoCondicoesIniciais := 30;
	
	//Passo 30 - Robô em Condições Iniciais
	30: 
		PassoCondicoesIniciais := 40;
		
	//Passo 40 - Servos X e Y em Condições Iniciais
	40:
		PassoCondicoesIniciais := 50;
		
	//Passo 50 - Mesa Index em Condições Iniciais
	50: 
		PassoCondicoesIniciais := 60;
		
	//Passo 60 - Câmera em Condições Iniciais
	60: 
		PassoCondicoesIniciais := 70;
		
	//Passo 70 - 
	70: 
		PassoCondicoesIniciais := 80;
	
	//Passo 80 - Sinalizar Conclusão da Rotina
	80: 
		PassoCondicoesIniciais := 1000;
	
	//Passo 1000 - Finalização
	1000: PassoCondicoesIniciais := 0;

END_CASE*)

(*========================================================================*)

END_PROGRAM

// ---- POUs/Alarmes.TcPOU
PROGRAM Alarmes
VAR

(*==========================		ALARMES		==========================*)
	TestBit							: BOOL;

	ByteAlarmeEmergencia			: BYTE;
	ByteAlarmeAberturaPortas		: BYTE;
	ByteAlarmePainelPneumatico		: BYTE;
	ByteAlarmeServoMotor			: BYTE;
	
	//AlarmeCortinaLuz				: BOOL;
	AlarmeEmergencia				: BOOL;
	AlarmeAberturaPortas			: BOOL;
	AlarmePainelPneumatico			: BOOL;
	AlarmeServoMotor				: BOOL;
	
	AlarmeGrave						: BOOL;
	AlarmeMedio						: BOOL;
	AlarmeLeve						: BOOL;

(*========================================================================*)

END_VAR

(*==========================		ALARMES		==========================*)

(*=====================		RESUMO DOS ALARMES		======================*)

IF (AlarmeEmergencia) THEN
	AlarmeGrave := TRUE;
ELSE
	AlarmeGrave := FALSE;
END_IF

IF (AlarmeAberturaPortas) THEN
	AlarmeMedio := TRUE;
ELSE
	AlarmeMedio := FALSE;
END_IF

IF (FALSE) THEN
	AlarmeLeve := TRUE;
ELSE
	AlarmeLeve := FALSE;
END_IF

(*========================================================================*) 

(*=================		ALARMES DE CORTINA DE LUZ		==================*)

//Alarme de Cortina de Luz
//IF (NOT InSafety_CortinaLuz) THEN
//	AlarmeCortinaLuz := TRUE;
//ELSIF (InSafety_CortinaLuz AND Reset) THEN
//	AlarmeCortinaLuz := FALSE;
//END_IF

(*========================================================================*) 

(*==================		ALARMES DE EMERGÊNCIA		==================*)

//Resumo do Byte
IF (ByteAlarmeEmergencia > 0) THEN
	AlarmeEmergencia := TRUE;
ELSE
	AlarmeEmergencia := FALSE;
END_IF

//Bit 0 - Botão de Emergência Frontal
IF (NOT InSafety_BtEmergenciaFrontal) THEN
	ByteAlarmeEmergencia.0 := TRUE;
ELSIF (InSafety_BtEmergenciaFrontal AND Reset) THEN
	ByteAlarmeEmergencia.0 := FALSE;
END_IF

//Bit 1 - Botão de Emergência do Chiller
IF (NOT InSafety_BtEmergenciaChiller) THEN
	ByteAlarmeEmergencia.1 := TRUE;
ELSIF (InSafety_BtEmergenciaChiller AND Reset) THEN
	ByteAlarmeEmergencia.1 := FALSE;
END_IF

//Bit 2 - Botão de Emergência da Porta Maq. Solda
IF (NOT InSafety_BtEmergenciaMaquinaSolda) THEN
	ByteAlarmeEmergencia.2 := TRUE;
ELSIF (InSafety_BtEmergenciaMaquinaSolda AND Reset) THEN
	ByteAlarmeEmergencia.2 := FALSE;
END_IF

//Bit 3 - Botão de Emergência do Robô
IF (NOT InSafety_BtEmergenciaRobo) THEN
	ByteAlarmeEmergencia.3	:= TRUE;
ELSIF (InSafety_BtEmergenciaRobo AND Reset) THEN
	ByteAlarmeEmergencia.3 := FALSE;
END_IF

(*========================================================================*) 

(*==================	ALARMES DE ABETURA DE PORTAS		==============*)

//Resumo do Byte
IF (ByteAlarmeAberturaPortas > 0) THEN
	AlarmeAberturaPortas := TRUE;
ELSE
	AlarmeAberturaPortas := FALSE;
END_IF

//Bit 0 - Abertura da Porta Frontal Inferior
IF (NOT InSafety_ChPortaFrontalInferior) THEN
	ByteAlarmeAberturaPortas.0 := TRUE;
ELSIF (InSafety_ChPortaFrontalInferior AND Reset) THEN
	ByteAlarmeAberturaPortas.0 := FALSE;
END_IF

//Bit 1 - Abertura da Porta da Câmera
IF (NOT InSafety_ChPortaCamera) THEN
	ByteAlarmeAberturaPortas.1 := TRUE;
ELSIF (InSafety_ChPortaCamera AND Reset) THEN
	ByteAlarmeAberturaPortas.1 := FALSE;
END_IF

//Bit 2 - Abertura da Porta da Esteira
IF (NOT InSafety_ChPortaEsteira) THEN
	ByteAlarmeAberturaPortas.2 := TRUE;
ELSIF (InSafety_ChPortaEsteira AND Reset) THEN
	ByteAlarmeAberturaPortas.2 := FALSE;
END_IF

//Bit 3 - Abertura da Porta Lateral Esquerda - Folha Direita
IF (NOT InSafety_ChPortaLateralEsquerdaFD) THEN
	ByteAlarmeAberturaPortas.3 := TRUE;
ELSIF (InSafety_ChPortaLateralEsquerdaFD AND Reset) THEN
	ByteAlarmeAberturaPortas.3 := FALSE;
END_IF

//Bit 4 - Abertura da Porta Lateral Esquerda - Folha Esquerda
IF (NOT InSafety_ChPortaLateralEsquerdaFE) THEN
	ByteAlarmeAberturaPortas.4 := TRUE;
ELSIF (InSafety_ChPortaLateralEsquerdaFE AND Reset) THEN
	ByteAlarmeAberturaPortas.4 := FALSE;
END_IF

//Bit 5 - Abertura da Porta da Máquina de Solda / Robô
IF (NOT InSafety_ChPortaMaquinaSolda) THEN
	ByteAlarmeAberturaPortas.5 := TRUE;
ELSIF (InSafety_ChPortaMaquinaSolda AND Reset) THEN
	ByteAlarmeAberturaPortas.5 := FALSE;
END_IF

//Bit 6 - Abertura da Porta do Painel Principal
IF (NOT InSafety_ChPortaPainelPrincipal) THEN
	ByteAlarmeAberturaPortas.6 := TRUE;
ELSIF (InSafety_ChPortaPainelPrincipal AND Reset) THEN
	ByteAlarmeAberturaPortas.6 := FALSE;
END_IF

(*========================================================================*) 

(*=================		ALARMES PAINEL PNEUMÁTICO		==================*)

//Resumo do Byte
IF (ByteAlarmePainelPneumatico > 0) THEN
	AlarmePainelPneumatico := TRUE;
ELSE
	AlarmePainelPneumatico := FALSE;
END_IF

//Bit 0 - Pressostato Geral (Digital)
IF (NOT InPressostatoGeral) THEN
	ByteAlarmePainelPneumatico.0 := TRUE;
	IhmVs_PressaoPainelPneumatico_Text	:= "Alarme de Pressão";
ELSIF (InPressostatoGeral AND Reset) THEN
	ByteAlarmePainelPneumatico.0 := FALSE;
	IhmVs_PressaoPainelPneumatico_Text	:= "Pressão Normal";
END_IF

//Bit 1 - Sensor Indutivo Válvula de Segurança V7
IF (InSensorSegValvY7) THEN
	ByteAlarmePainelPneumatico.1 := TRUE;
ELSIF (NOT InSensorSegValvY7 AND Reset) THEN
	ByteAlarmePainelPneumatico.1 := FALSE;
END_IF

//Bit 2 - Sensor Indutivo Válvula de Segurança V8
IF (InSensorSegValvY8) THEN
	ByteAlarmePainelPneumatico.2 := TRUE;
ELSIF (NOT InSensorSegValvY8 AND Reset) THEN
	ByteAlarmePainelPneumatico.2 := FALSE;
END_IF

(*========================================================================*)

(*=================		ALARMES SERVO MOTORES X E Y		==================*)

//Resumo do Byte
IF (ByteAlarmeServoMotor > 0) THEN
	AlarmeServoMotor := TRUE;
ELSE
	AlarmeServoMotor := FALSE;
END_IF

//Bit 0 - 
IF (NOT InPressostatoGeral) THEN
	ByteAlarmePainelPneumatico.0 := TRUE;
ELSIF (InPressostatoGeral AND Reset) THEN
	ByteAlarmePainelPneumatico.0 := FALSE;
END_IF
(*========================================================================*)

END_PROGRAM

// ---- POUs/InterfaceIOs.TcPOU
PROGRAM InterfaceIOs
VAR
END_VAR

(*======================		ENTRADAS DIGITAIS		======================*)

	//Cartão de Entradas 0:= EntradaI0_0
	InMaquinaSolda_FK		:= EntradaI0_0;
//	InPinoCalha				:= EntradaI0_1;
//	InReset					:= EntradaI0_2;
//	InVermelho				:= EntradaI0_3;
//	InAmarelo				:= EntradaI0_4;
//	InVerde					:= EntradaI0_5;
//	InPecaOK				:= EntradaI0_6;
//	InSolda					:= EntradaI0_7;
	InFimCurso1				:= EntradaI1_0;
	InFimCurso2				:= EntradaI1_1;
	InFimCurso3				:= EntradaI1_2;
	InFimCurso4				:= EntradaI1_3;
//	InSensorIndutivo01		:= EntradaI1_4;
//	InSensorIndutivo02		:= EntradaI1_5;
//	InSensorIndutivo03		:= EntradaI1_6;
//	InSensorIndutivo04		:= EntradaI1_7;
	
	//Cartão de Entradas 1
//	InSensorIndutivo05		:= EntradaI2_0;
//	InSensorIndutivo06		:= EntradaI2_1;
	InSensorIndutivo07		:= EntradaI2_2;
//	InSensorIndutivo08		:= EntradaI2_3;
//	InSensorIndutivo09		:= EntradaI2_4;
//	InSensorIndutivo10		:= EntradaI2_5;
//	InSensorIndutivo11		:= EntradaI2_6;
//	InSensorIndutivo12		:= EntradaI2_7;
//	InComandoX				:= EntradaI3_0;
//	InComandoY				:= EntradaI3_1;
//	InComandoZ				:= EntradaI3_2;
//	InComando4				:= EntradaI3_3;
//	InComando5				:= EntradaI3_4;
//	InComando6				:= EntradaI3_5;
//	InComandoX1				:= EntradaI3_6;
//	InComandoX10			:= EntradaI3_7;
	
	//Cartão de Entradas 2
//	InComandoX100			:= EntradaI4_0;
//	Reserva					:= EntradaI4_1;
//	Reserva					:= EntradaI4_2;
//	Reserva					:= EntradaI4_3;
//	Reserva					:= EntradaI4_4;
//	Reserva					:= EntradaI4_5;
//	Reserva					:= EntradaI4_6;
//	Reserva					:= EntradaI4_7;
//	InSinalFaltaFase		:= EntradaI5_0;
//	InComandoPedal			:= EntradaI5_1;
	InSolicitaEntrada		:= EntradaI5_2;
	InSolicitaReset			:= EntradaI5_3;
//	Reserva					:= EntradaI5_4;
//	Reserva					:= EntradaI5_5;
//	Reserva					:= EntradaI5_6;
//	Reserva					:= EntradaI5_7;
	
	//Cartão de Entradas 3
	InPressostatoGeral		:= EntradaI6_0;
	InSensorSegValvY7		:= EntradaI6_1;
	InSensorSegValvY8		:= EntradaI6_2;
//	InPeçaGarraRobo			:= EntradaI6_3;
//	Reserva					:= EntradaI6_4;
//	Reserva					:= EntradaI6_5;
//	Reserva					:= EntradaI6_6;
//	Reserva					:= EntradaI6_7;
//	Reserva					:= EntradaI7_0;
//	Reserva					:= EntradaI7_1;
//	Reserva					:= EntradaI7_2;
//	Reserva					:= EntradaI7_3;
//	Reserva					:= EntradaI7_4;
//	Reserva					:= EntradaI7_5;
//	Reserva					:= EntradaI7_6;
//	Reserva					:= EntradaI7_7;
		
(*============================================================================*)

(*=========================		SAÍDAS DIGITAIS		==========================*)
	//Outputs
	
	//Cartão de Saídas 0
	SaidaQ0_0				:= OutLigarMesaIndex;
	SaidaQ0_1				:= OutSentidoGiroMesaIndex;
	SaidaQ0_2				:= OutLigarEsteiraSaida;
	SaidaQ0_3				:= OutSentidoGiroEsteiraSaida;
	SaidaQ0_4				:= OutMaquinaSolda_BtReset;
	SaidaQ0_5				:= OutMaquinaSolda_BtStart;
//	SaidaQ0_6				:= OutMaquinaSolda_BtReserva;
	SaidaQ0_7				:= OutMaquinaSolda_Receita_Bit1;
	SaidaQ1_0				:= OutMaquinaSolda_Receita_Bit2;
	SaidaQ1_1				:= OutMaquinaSolda_Receita_Bit3;
	SaidaQ1_2				:= OutMaquinaSolda_Receita_Bit4;
	SaidaQ1_3				:= OutMaquinaSolda_Receita_Bit5;
//	SaidaQ1_4				:= OutMaquinaSolda_Reserva;
//	SaidaQ1_5				:= OutMaquinaSolda_Reserva;
//	SaidaQ1_6				:= OutMaquinaSolda_Reserva;
	SaidaQ1_7				:= OutValvulaY1A;
	
	//Cartão de Saídas 1
	SaidaQ2_0				:= OutValvulaY1R;
//	SaidaQ2_1				:= OutValvulaY2A;
//	SaidaQ2_2				:= OutValvulaY2R;
//	SaidaQ2_3				:= OutValvulaY3A;
//	SaidaQ2_4				:= OutValvulaY3R;
//	SaidaQ2_5				:= OutValvulaY4A;
//	SaidaQ2_6				:= OutValvulaY4R;
	SaidaQ2_7				:= OutValvulaY5A;
	SaidaQ3_0				:= OutValvulaY5R;
	SaidaQ3_1				:= OutValvulaY6;
	SaidaQ3_2				:= OutValvulaY7;
	SaidaQ3_3				:= OutValvulaY8;
	SaidaQ3_4				:= OutValvulaY9;
//	SaidaQ3_5				:= OutSinalizadorComandoLigado;
	SaidaQ3_6				:= OutSinalizadorBotoeiraHS1;
	SaidaQ3_7				:= OutSinalizadorBotoeiraHS2;
	
	//Cartão de Saídas 2
	//SaidaQ4_0				:= ;
	//SaidaQ4_1				:= ;
	//SaidaQ4_2				:= ;
	//SaidaQ4_3				:= ;
	//SaidaQ4_4				:= ;
	//SaidaQ4_5				:= ;
	//SaidaQ4_6				:= ;
	//SaidaQ4_7				:= ;
	//SaidaQ5_0				:= ;
	//SaidaQ5_1				:= ;
	//SaidaQ5_2				:= ;
	//SaidaQ5_3				:= ;
	//SaidaQ5_4				:= ;
	//SaidaQ5_5				:= ;
	//SaidaQ5_6				:= ;
	//SaidaQ5_7				:= ;
	
	//Cartão de Saídas 3
	//SaidaQ6_0				:= ;
	//SaidaQ6_1				:= ;
	//SaidaQ6_2				:= ;
	//SaidaQ6_3				:= ;
	//SaidaQ6_4				:= ;
	//SaidaQ6_5				:= ;
	//SaidaQ6_6				:= ;
	//SaidaQ6_7				:= ;
	//SaidaQ7_0				:= ;
	//SaidaQ7_1				:= ;
	//SaidaQ7_2				:= ;
	//SaidaQ7_3				:= ;
	//SaidaQ7_4				:= ;
	//SaidaQ7_5				:= ;
	//SaidaQ7_6				:= ;
	//SaidaQ7_7				:= ;

(*============================================================================*)

(*======================		ENTRADAS ANALÓGICAS		======================*)	
	
	ReguaPotenciometricaSinal	:= EntradaA0_0;
	//							:= EntradaA0_1;
	//							:= EntradaA0_2;
	//							:= EntradaA0_3;
	
(*============================================================================*)

(*======================		SAÍDAS ANALÓGICAS		======================*)

	SaidaA0_0				:= REAL_TO_INT(ValvulaProporcional);
	SaidaA0_1				:= REAL_TO_INT(FrequenciaMesaIndex);
	SaidaA0_2				:= REAL_TO_INT(FrequenciaEsteiraSaida);
//	SaidaA0_2				:= ;

(*============================================================================*)

(*==========================		SAFETY PLC		==========================*)	

	InSafety_CortinaLuz					:= SafetyPLC_In_Byte0.0;
	InSafety_BtEmergenciaMaquinaSolda	:= SafetyPLC_In_Byte0.2;
	InSafety_BtEmergenciaChiller		:= SafetyPLC_In_Byte1.4;
	InSafety_BtEmergenciaRobo			:= SafetyPLC_In_Byte1.6;
	InSafety_BtEmergenciaFrontal		:= SafetyPLC_In_Byte2.0;
	InSafety_ChPortaMaquinaSolda		:= SafetyPLC_In_Byte0.4;
	InSafety_ChPortaPainelPrincipal		:= SafetyPLC_In_Byte0.6;
	InSafety_ChPortaEsteira				:= SafetyPLC_In_Byte1.0;
	InSafety_ChPortaCamera				:= SafetyPLC_In_Byte1.2;
	InSafety_ChPortaFrontalInferior		:= SafetyPLC_In_Byte2.2;
	InSafety_ChPortaLateralEsquerdaFD	:= SafetyPLC_In_Byte2.4;
	InSafety_ChPortaLateralEsquerdaFE	:= SafetyPLC_In_Byte2.6;
	
	OutSafety_LiberacaoSDV1				:= SafetyPLC_In_Byte3.0;
	OutSafety_ComandoSDV1				:= SafetyPLC_In_Byte3.1;
	OutSafety_LiberacaoSDV2				:= SafetyPLC_In_Byte3.2;
	OutSafety_ComandoSDV2				:= SafetyPLC_In_Byte3.3;
	OutSafety_ComandoINVMesaIndex		:= SafetyPLC_In_Byte4.0;
	OutSafety_ComandoINVEsteiraSaida	:= SafetyPLC_In_Byte4.1;
	OutSafety_Comando1Robo				:= SafetyPLC_In_Byte4.2;
	OutSafety_Comando2Robo				:= SafetyPLC_In_Byte4.3;
	OutSafety_ParadaMaquinaSolda		:= SafetyPLC_In_Byte5.0;
	OutSafety_SinalizacaoEmergencia		:= SafetyPLC_In_Byte5.1;
	OutSafety_Reserva1					:= SafetyPLC_In_Byte5.2;
	OutSafety_Reserva2					:= SafetyPLC_In_Byte5.3;
	
	SafetyPLC_Out_Byte0.0				:= Reset;//OutSafety_BtReset;
	
(*============================================================================*)

END_PROGRAM

// ---- POUs/Perifericos/Inversores.TcPOU
PROGRAM Inversores
VAR

(*=========================		INVERSORES		==========================*)	

	PassoMesaIndexAutomatico		: INT;
	PassoMesaIndexCiclo				: INT;
	PassoMesaIndexFwd				: INT;
	PassoMesaIndexBwd				: INT;
	PassoEsteiraSaidaAutomatico		: INT;
	PassoEsteiraSaidaFwd			: INT;
	PassoEsteiraSaidaBwd			: INT;

	TON_DelayParadaAuto				: TON;
	TON_DelayParadaCiclo			: TON;
	
	DelayParada						: TIME;
	
(*========================================================================*)

END_VAR

(*==============		SET Velocidade da Mesa Index		==============*)

FrequenciaMesaIndex := (INT_TO_REAL(IhmEscr_MesaIndex_Frequencia)/60)*(32767);
DelayParada	:= REAL_TO_TIME(IhmEscr_MesaIndex_DelayParada*1000);

(*=================		INVERSOR 1 - Mesa Index		======================*)

(*======================		Modo Automático		======================*)

//Condição de Bloqueio da Máquina de Estados - Mesa Index Automático
IF (Alarmes.AlarmeGrave
	//OR Alarmes.AlarmeMedio
	//OR Alarmes.AlarmeLeve
	OR NOT MaquinaLigada
	OR NOT MaquinaModoAuto
	OR NOT((ReguaPotenciometricaPosicao > ReguaPotenciometrica_Recuada_LI) AND (ReguaPotenciometricaPosicao < ReguaPotenciometrica_Recuada_LS))
	OR (NOT InSafety_CortinaLuz AND (PassoMesaIndexAutomatico > 13))
	) THEN
	PassoMesaIndexAutomatico := 1000;
	TON_DelayParadaAuto(IN:=FALSE);
	Flag_MesaIndex_Maquina := FALSE;
	LigarMesaIndexAutomatico := FALSE;	
END_IF

CASE PassoMesaIndexAutomatico OF
	
	//Passo 0 - Inicialização	
	0: PassoMesaIndexAutomatico := 10;
	
	//Passo 10 - Condição para Iniciar a Rotina Mesa Index (Sentido Normal - Automatico)
	10: IF  (Flag_Maquina_MesaIndex) THEN
			Flag_Maquina_MesaIndex := FALSE;
			PassoMesaIndexAutomatico := 11;
		END_IF

	//Passo 11 - Barreira Livre - Início do Processo
	11: IF  (InSafety_CortinaLuz) THEN
			PassoMesaIndexAutomatico := 12;
		END_IF
		
	//Passo 12 - Barreira Rompida - Posicionar Peça
	12: IF  (NOT InSafety_CortinaLuz) THEN
			PassoMesaIndexAutomatico := 13;
		END_IF
		
	//Passo 13 - Barreira Livre - Iniciar Movimentação da Mesa
	13: IF  (InSafety_CortinaLuz) THEN
			PassoMesaIndexAutomatico := 14;
		END_IF
		
	//Passo 14 - Movimentar Mesa Index
	14: LigarMesaIndexAutomatico := TRUE;
		
		Flag_Maquina_MesaIndex := FALSE;//Fora de posição para efeito de testes
	
		PassoMesaIndexAutomatico := 20;

	//Passo 20 - Aguardar Acionamento do Sensor de Posição 
	20: IF  InSensorIndutivo07 THEN
			PassoMesaIndexAutomatico := 30;	
		END_IF
	
	//Passo 30 - Aguardar Desacionamento do Sensor de Posição 
	30: IF  NOT InSensorIndutivo07 THEN
			PassoMesaIndexAutomatico := 40;	
		END_IF	

	//Passo 40 - Condição para Desligar Mesa Index - Delay de Parada
	40: TON_DelayParadaAuto(IN:=TRUE,PT:= DelayParada);
		IF (TON_DelayParadaAuto.Q) THEN
			TON_DelayParadaAuto(IN:=FALSE);
			LigarMesaIndexAutomatico := FALSE;
			PassoMesaIndexAutomatico := 50;
		END_IF
	
	//Passo 50 - Sinalização da Conclusão do Movimento
	50: Flag_MesaIndex_Maquina := TRUE;
		PassoMesaIndexAutomatico := 1000;
			
	//Passo 1000 - Finalização
	1000: PassoMesaIndexAutomatico := 0;
	
END_CASE

(*========================================================================*)

(*=========================		Modo Ciclo		==========================*)

//Condição de Bloqueio da Máquina de Estados - Mesa Index Ciclo
IF (Alarmes.AlarmeGrave 
	OR NOT MaquinaModoManual
	OR NOT InSafety_CortinaLuz
	) THEN
	PassoMesaIndexCiclo := 1000;
	TON_DelayParadaCiclo(IN:=FALSE);
	LigarMesaIndexCiclo := FALSE;
END_IF

CASE PassoMesaIndexCiclo OF
	
	//Passo 0 - Inicialização	
	0: PassoMesaIndexCiclo := 10;
	
	//Passo 10 - Condição para Ligar Mesa Index (Sentido Normal - Ciclo)
	10: IF  (IhmBt_MesaIndex_Ciclo) THEN
			PassoMesaIndexCiclo := 20;
		END_IF
		
	//Passo 20 - Aguardar o Botão Retorno do Botão
	20: IF  (NOT IhmBt_MesaIndex_Ciclo) THEN
			PassoMesaIndexCiclo := 30;
		END_IF
 
	//Passo 30 - Ligar Mesa Index
	30: LigarMesaIndexCiclo := TRUE;
		IF (InSensorIndutivo07) THEN
			PassoMesaIndexCiclo := 40;	
		END_IF
		
	//Passo 40 - Aguardar Desacionamento do Sensor de Posição 
	40:	IF (NOT InSensorIndutivo07) THEN
			PassoMesaIndexCiclo := 50;	
		END_IF

	//Passo 50 - Condição para Desligar Mesa Index 
	50: TON_DelayParadaCiclo(IN:=TRUE,PT:= DelayParada);
		IF (TON_DelayParadaCiclo.Q) THEN
			TON_DelayParadaCiclo(IN:=FALSE);
			LigarMesaIndexCiclo := FALSE;
			PassoMesaIndexCiclo := 1000;
		END_IF
			
	//Passo 1000 - Finalização
	1000: PassoMesaIndexCiclo := 0;
	
END_CASE

(*========================================================================*)

(*======================		Modo Manual		==========================*)

//Condição de Bloqueio da Máquina de Estados - Mesa Index FWD
IF (Alarmes.AlarmeGrave
	OR NOT MaquinaModoManual
	OR(NOT IhmBt_MesaIndex_LigarDesligar AND IhmBt_MesaIndex_Sentido)
	OR IhmBt_MesaIndex_Ciclo
	OR NOT InSafety_CortinaLuz
	) THEN
	PassoMesaIndexFwd := 1000;
	LigarMesaIndexFwd := FALSE;
	IhmBt_MesaIndex_LigarDesligar := FALSE;
END_IF

CASE PassoMesaIndexFwd OF
	
	//Passo 0 - Inicialização	
	0: PassoMesaIndexFwd := 10;
	
	//Passo 10 - Condição para Ligar Mesa Index (Sentido Normal - Forward)
	10: IF (NOT IhmBt_MesaIndex_Sentido AND IhmBt_MesaIndex_LigarDesligar) THEN
			LigarMesaIndexFwd := TRUE;
			PassoMesaIndexFwd := 20;
		END_IF

	//Passo 20 - Condição para Desligar Mesa Index 
	20: IF (NOT IhmBt_MesaIndex_LigarDesligar) THEN
			LigarMesaIndexFwd := FALSE;
			PassoMesaIndexFwd := 1000;	
		END_IF
	
	//Passo 1000 - Finalização
	1000: PassoMesaIndexFwd := 0;
	
END_CASE

//Condição de Bloqueio da Máquina de Estados - Mesa Index REV
IF (Alarmes.AlarmeGrave
	//OR NOT MaquinaModoManual
	//OR(NOT IhmBt_MesaIndex_LigarDesligar AND NOT IhmBt_MesaIndex_Sentido)
	OR IhmBt_MesaIndex_Ciclo
	) THEN
	PassoMesaIndexBwd := 1000;
	LigarMesaIndexBwd := FALSE;
	IhmBt_MesaIndex_LigarDesligar := FALSE;
END_IF

CASE PassoMesaIndexBwd OF
	
	//Passo 0 - Inicialização	
	0: PassoMesaIndexBwd := 10;
	
	//Passo 10 - Condição para Ligar Mesa Index (Sentido Reverso - Reverse)
	10: IF (IhmBt_MesaIndex_Sentido AND IhmBt_MesaIndex_LigarDesligar) THEN
			LigarMesaIndexBwd := TRUE;
			PassoMesaIndexBwd := 20;
		END_IF

	//Passo 20 - Condição para Desligar Mesa Index 
	20: IF (NOT IhmBt_MesaIndex_LigarDesligar) THEN
			LigarMesaIndexBwd := FALSE;
			PassoMesaIndexBwd := 1000;	
		END_IF
	
	//Passo 1000 - Finalização
	1000: PassoMesaIndexBwd := 0;
	
END_CASE

(*=============		SET Velocidade da Esteira de Saída		==============*)

FrequenciaEsteiraSaida := (INT_TO_REAL(IhmEscr_EsteiraSaida_Frequencia)/60)*(32767);

(*=============		INVERSOR 2 - Esteira de Saída		==================*)

(*======================		Modo Automático		======================*)



(*======================		Modo Manual		==========================*)

//Condição de Bloqueio da Máquina de Estados - Esteira de Saída FWD
IF (Alarmes.AlarmeGrave
	OR NOT MaquinaModoManual
	OR(NOT IhmBt_EsteiraSaida_LigarDesligar AND IhmBt_EsteiraSaida_Sentido)
	) THEN
	PassoEsteiraSaidaFwd := 1000;
	LigarEsteiraSaidaFwd := FALSE;
END_IF

CASE PassoEsteiraSaidaFwd OF
	
	//Passo 0 - Inicialização	
	0: PassoEsteiraSaidaFwd := 10;
	
	//Passo 10 - Condição para Ligar Esteira de Saída (Sentido Normal - Forward)
	10: IF (NOT IhmBt_EsteiraSaida_Sentido AND IhmBt_EsteiraSaida_LigarDesligar) THEN
			LigarEsteiraSaidaFwd := TRUE;
			PassoEsteiraSaidaFwd := 20;
		END_IF

	//Passo 20 - Condição para Desligar Esteira de Saída 
	20: IF (NOT IhmBt_EsteiraSaida_LigarDesligar) THEN
			LigarEsteiraSaidaFwd := FALSE;
			PassoEsteiraSaidaFwd := 1000;	
		END_IF
	
	//Passo 1000 - Finalização
	1000: PassoEsteiraSaidaFwd := 0;
	
END_CASE

//Condição de Bloqueio da Máquina de Estados - Esteira de Saída REV
IF (Alarmes.AlarmeGrave
	//OR NOT MaquinaModoManual
	OR(NOT IhmBt_EsteiraSaida_LigarDesligar AND NOT IhmBt_EsteiraSaida_Sentido)
	) THEN
	PassoEsteiraSaidaBwd := 1000;
	LigarEsteiraSaidaBwd := FALSE;		
END_IF

CASE PassoEsteiraSaidaBwd OF
	
	//Passo 0 - Inicialização	
	0: PassoEsteiraSaidaBwd := 10;
	
	//Passo 10 - Condição para Ligar Mesa Index (Sentido Reverso - Reverse)
	10: IF (IhmBt_EsteiraSaida_Sentido AND IhmBt_EsteiraSaida_LigarDesligar) THEN
			LigarEsteiraSaidaBwd := TRUE;
			PassoEsteiraSaidaBwd := 20;
		END_IF

	//Passo 20 - Condição para Desligar Mesa Index 
	20: IF (NOT IhmBt_EsteiraSaida_LigarDesligar) THEN
			LigarEsteiraSaidaBwd := FALSE;
			PassoEsteiraSaidaBwd := 1000;	
		END_IF
	
	//Passo 1000 - Finalização
	1000: PassoEsteiraSaidaBwd := 0;
	
END_CASE

(*========================================================================*)

(*=====================		INVERSORES	- SAÍDAS	======================*)	

//Inversor 1 - Mesa Index
IF (LigarMesaIndexFwd OR LigarMesaIndexCiclo OR LigarMesaIndexAutomatico) THEN
	OutSentidoGiroMesaIndex := FALSE;
	OutLigarMesaIndex := TRUE;
ELSIF (LigarMesaIndexBwd) THEN
	OutSentidoGiroMesaIndex := TRUE;
	OutLigarMesaIndex := TRUE;
ELSE
	OutSentidoGiroMesaIndex := FALSE;
	OutLigarMesaIndex := FALSE;
END_IF

//Inversor 2 - Esteira de Saída
IF (LigarEsteiraSaidaFwd) THEN
	OutSentidoGiroEsteiraSaida := FALSE;
	OutLigarEsteiraSaida := TRUE;
ELSIF (LigarEsteiraSaidaBwd) THEN
	OutSentidoGiroEsteiraSaida := TRUE;
	OutLigarEsteiraSaida := TRUE;
ELSE
	OutSentidoGiroEsteiraSaida := FALSE;
	OutLigarEsteiraSaida := FALSE;
END_IF

(*========================================================================*)

END_PROGRAM

// ---- POUs/Perifericos/Valvulas.TcPOU
PROGRAM Valvulas
VAR

(*=========================		VÁLVULAS		==========================*)	



(*========================================================================*)

END_VAR

(*==============		Válvula Y1 - XXXXXXX XXXXXXX		==============*)

IF (MaquinaModoManual) THEN
	//Controle Manual - Válvula Y1
	IF (IhmBt_Y1_Ligar) THEN
		OutValvulaY1R := FALSE;	//Solenóide de Recuo
		OutValvulaY1A := TRUE; //Solenóide de Avanço
	ELSE
		OutValvulaY1A := FALSE;	//Solenóide de Avanço
		OutValvulaY1R := TRUE; //Solenóide de Recuo	
	END_IF
ELSIF (MaquinaModoAuto) THEN
	//Controle Automático - Válvula Y1
	IF (AvancarValvulaY1) THEN
		OutValvulaY1R := FALSE; //Solenóide de Recuo
		OutValvulaY1A := TRUE;	//Solenóide de Avanço
	ELSE
		OutValvulaY1A := FALSE; //Solenóide de Avanço
		OutValvulaY1R := TRUE;	//Solenóide de Recuo
	END_IF
ELSE
	OutValvulaY1R := FALSE; //Solenóide de Recuo
	OutValvulaY1A := FALSE;	//Solenóide de Avanço
END_IF

(*========================================================================*)

(*==============		Válvula Y2 - XXXXXXX XXXXXXX		==============*)

IF (MaquinaModoManual) THEN
	//Controle Manual - Válvula Y2
	IF (IhmBt_Y2_Ligar) THEN
		OutValvulaY2R := FALSE;	//Solenóide de Recuo
		OutValvulaY2A := TRUE; //Solenóide de Avanço
	ELSE
		OutValvulaY2A := FALSE;	//Solenóide de Avanço
		OutValvulaY2R := TRUE; //Solenóide de Recuo	
	END_IF
ELSIF (MaquinaModoAuto) THEN
	//Controle Automático - Válvula Y2
	IF (AvancarValvulaY2) THEN
		OutValvulaY2R := FALSE; //Solenóide de Recuo
		OutValvulaY2A := TRUE;	//Solenóide de Avanço
	ELSE
		OutValvulaY2A := FALSE; //Solenóide de Avanço
		OutValvulaY2R := TRUE;	//Solenóide de Recuo
	END_IF
ELSE
	OutValvulaY2R := FALSE; //Solenóide de Recuo
	OutValvulaY2A := FALSE;	//Solenóide de Avanço
END_IF

(*========================================================================*)

(*==============		Válvula Y3 - XXXXXXX XXXXXXX		==============*)

IF (MaquinaModoManual) THEN
	//Controle Manual - Válvula Y3
	IF (IhmBt_Y3_Ligar) THEN
		OutValvulaY3R := FALSE;	//Solenóide de Recuo
		OutValvulaY3A := TRUE; //Solenóide de Avanço
	ELSE
		OutValvulaY3A := FALSE;	//Solenóide de Avanço
		OutValvulaY3R := TRUE; //Solenóide de Recuo	
	END_IF
ELSIF (MaquinaModoAuto) THEN
	//Controle Automático - Válvula Y3
	IF (AvancarValvulaY3) THEN
		OutValvulaY3R := FALSE; //Solenóide de Recuo
		OutValvulaY3A := TRUE;	//Solenóide de Avanço
	ELSE
		OutValvulaY3A := FALSE; //Solenóide de Avanço
		OutValvulaY3R := TRUE;	//Solenóide de Recuo
	END_IF
ELSE
	OutValvulaY3R := FALSE; //Solenóide de Recuo
	OutValvulaY3A := FALSE;	//Solenóide de Avanço
END_IF

(*========================================================================*)

(*==============		Válvula Y4 - XXXXXXX XXXXXXX		==============*)

